# B&R Automation Studio project TD52 (part 60)

#### Gen2_ref.c
```c
/********************************************************************
 * COPYRIGHT -- B&R Industrial Automation GmbH
 ********************************************************************
 * Program: Gen2_ref
 * File: Gen2_ref.c
 * Author: 105055527
 * Last modified by: kelleto00
 * Created: Wed Apr 16 13:02:53 2008
 * Last modified: Wed Oct 09 10:01:33 2024
 * Model Version: 4.14.00.04
 * Description: V4.10.00.01, 01-09-2020 Keller, Ke Estimator, additive LS factor, Ptraj SpeedCtrl, LVRT Freeze HLCi
   V4.10.00.01, 02-10-2020 Keller, bugfix HLCi p2srefLX init, BDC_lib: change Inf to 1e7
   V4.10.00.01, 13-11-2020 Keller, bugfix LXcorr T2s/ZZP, LSLff damping, dbgOut for Leanox WG compensation
   V4.10.00.01, 27-01-2021 Keller, Lx WGV compensation: no reset in island mode, addition before skipfire compensation
   V4.10.00.01, 02-02-2021 Keller, initialization lambda estimation with rLam_Start
   V4.11.00.01, 28-05-2021 Keller, Gas Quality Change (GQC) Improvements, LHV estimator output
   V4.11.00.01, 05-11-2021 Keller, Bugfix BDC: worksplit offset, optionally Nset instead of Nnom, rN_Eng_LRskipF
   V4.12.00.01, 10-02-2021 Keller, SpeedCtrl2.0 TU Wien: Disturbance Estimator, LQR incl. droop & leanox
   V4.12.00.02, 23-05-2022 Arnold, Leanox point C in low load
   V4.12.00.02, 09-06-2022 Kafka, add external skip fire input for isolated and grid parallel operation
   V4.12.00.03, 15-09-2022 Keller, add power trajectory to HLCi for extended LQR (Droop setpoint)
   V4.12.00.04, 12-10-2022 Keller, add gas flow comp. factor for rejections
   V4.12.00.05, 13-10-2022 Keller, power filter for static skipfire in island mode
   V4.12.00.06, 15-11-2022 Keller, Ke adaptation with disturbance observer
   V4.13.00.01, 15-11-2022 Keller, FDC: R_mix output, HLCi: R_mix for Ke
   V4.13.00.02, 10-07-2023 Keller, interpolation of LHV, rho_gas and Lmin
   V4.13.00.03, 10-07-2023 Keller, load dependent gas dosage delay
   V4.13.00.04, 11-09-2023 Keller, D-part FSM, bugfix dPTV ramp
   V4.13.00.05, 27-02-2024 Keller, Filter outputs without bSS
   V4.13.00.06, 10-04-2024 Keller, bugfix leanox manual mode with bSepEmisCtrl
   V4.14.00.01, 01-07-2024 Keller, iNskip_LRfor Ke calculation
   V4.14.00.02, 17-09-2024 Keller, Use actual speed for observer disturbance dg (Gen2_ref/HLC_Island (HLC_Island_ref)/iLQR_SF/Ref LQR)
   V4.14.00.03, 30-09-2024 Keller, LR gas flow compensation possible without actuator saturation
   V4.14.00.04, 02-10-2024 Keller, Limit derivative power setpoint for FSM
 * modified Comment:
 ********************************************************************
 * Implementation of program Gen2_ref
 ********************************************************************
 * Generated with B&R Automation Studio Target for Simulink V6.7.1
 * (ERT based)
 ********************************************************************/

#include "Gen2_ref.h"
#include "Gen2_ref_private.h"

/*  Defines */

/*  Data Types */

/**************************** GLOBAL DATA *************************************/
/*  Definitions */

/*  Declarations  */

/* Forward declaration for local functions */
static real_T Gen2_ref_maximum(const real_T x[13], struct Gen2* inst);

/* Forward declaration for local functions */
static real_T Gen2_ref_minimum(const real_T x[13], struct Gen2* inst);
static real_T Gen2_ref_maximum_f(const real_T x[13], struct Gen2* inst);
static void Gen2_ref_diag(const real_T v[2], real_T d[4], struct Gen2* inst);
static void Gen2_ref_diag_i(const real_T v[4], real_T d[16], struct Gen2* inst);
static void Gen2_ref_diag_i2(const real_T v[3], real_T d[9], struct Gen2* inst);
static void Gen2_ref_state_space_d(const real_T x[3], const real_T p[22], real_T
  Ke_in, real_T Phi[9], real_T h[12], real_T hd[3], struct Gen2* inst);
static void Gen2_ref_diag_i2a(const real_T v[6], real_T d[36], struct Gen2* inst);
static real_T Gen2_ref_det(const real_T x[9], struct Gen2* inst);
static void Gen2_ref_mrdiv(const real_T A[18], const real_T B[9], real_T Y[18], struct Gen2* inst);
static void Gen2_ref_mldivide(const real_T A[16], const real_T B[12], real_T Y
  [12], struct Gen2* inst);
static void Gen2_ref_integrate_model(real_T x0[3], const real_T K[12], const
  real_T u2_past[100], real_T d, const real_T x_disturb[3], const real_T Bd[9],
  real_T x_disturb1_map, const real_T u_sp[4], const real_T x_sp[3], int16_T N,
  const real_T u_min[4], const real_T u_max[4], const real_T p[22], struct Gen2* inst);
static void Gen2_ref_mldivide_j(const real_T A[4], const real_T B[12], real_T Y
  [12], struct Gen2* inst);
static real_T Gen2_ref_maximum_f5(const real_T x[7], struct Gen2* inst);

/***************************** FILE SCOPE DATA ********************************/

/*************************** FUNCTIONS ****************************************/

/* Lookup Binary Search Utility BINARYSEARCH_real_T */
void BINARYSEARCH_real_T(uint32_T *piLeft, uint32_T *piRght, real_T u, const
  real_T *pData, uint32_T iHi, struct Gen2* inst)
{
  /* Find the location of current input value in the data table. */
  *piLeft = 0U;
  *piRght = iHi;
  if (u <= pData[0] ) {
    /* Less than or equal to the smallest point in the table. */
    *piRght = 0U;
  } else if (u >= pData[iHi] ) {
    /* Greater than or equal to the largest point in the table. */
    *piLeft = iHi;
  } else {
    uint32_T i;

    /* Do a binary search. */
    while (( *piRght - *piLeft ) > 1U ) {
      /* Get the average of the left and right indices using to Floor rounding. */
      i = (*piLeft + *piRght) >> 1;

      /* Move either the right index or the left index so that */
      /*  LeftDataPoint <= CurrentValue < RightDataPoint */
      if (u < pData[i] ) {
        *piRght = i;
      } else {
        *piLeft = i;
      }
    }
  }
}

/* Lookup Utility LookUp_real_T_real_T */
void LookUp_real_T_real_T(real_T *pY, const real_T *pYData, real_T u, const
  real_T *pUData, uint32_T iHi, struct Gen2* inst)
{
  uint32_T iLeft;
  uint32_T iRght;
  BINARYSEARCH_real_T( &(iLeft), &(iRght), u, pUData, iHi, inst);

  {
    real_T lambda;
    if (pUData[iRght] > pUData[iLeft] ) {
      real_T num;
      real_T den;
      den = pUData[iRght];
      den -= pUData[iLeft];
      num = u;
      num -= pUData[iLeft];
      lambda = num / den;
    } else {
      lambda = 0.0;
    }

    {
      real_T yLeftCast;
      real_T yRghtCast;
      yLeftCast = pYData[iLeft];
      yRghtCast = pYData[iRght];
      yLeftCast += lambda * ( yRghtCast - yLeftCast );
      (*pY) = yLeftCast;
    }
  }
}

/* Lookup Utility LookUp_real_T_real_T_SAT */
void LookUp_real_T_real_T_SAT(real_T *pY, const real_T *pYData, real_T u, const
  real_T *pUData, uint32_T iHi, struct Gen2* inst)
{
  uint32_T iLeft;
  uint32_T iRght;
  BINARYSEARCH_real_T( &(iLeft), &(iRght), u, pUData, iHi, inst);

  {
    real_T lambda;
    if (pUData[iRght] > pUData[iLeft] ) {
      real_T num;
      real_T den;
      den = pUData[iRght];
      den -= pUData[iLeft];
      num = u;
      num -= pUData[iLeft];
      lambda = num / den;
    } else {
      lambda = 0.0;
    }

    {
      real_T yLeftCast;
      real_T yRghtCast;
      yLeftCast = pYData[iLeft];
      yRghtCast = pYData[iRght];
      yLeftCast += lambda * ( yRghtCast - yLeftCast );
      (*pY) = yLeftCast;
    }
  }
}

/* Lookup Utility LookUp_real_Treal32_T_K4km1JJi */
void LookUp_real_Treal32_T_K4km1JJi(real_T *pY, const real32_T *pYData, real_T
  u, const real_T *pUData, uint32_T iHi, struct Gen2* inst)
{
  uint32_T iLeft;
  uint32_T iRght;
  BINARYSEARCH_real_T( &(iLeft), &(iRght), u, pUData, iHi, inst);

  {
    real_T lambda;
    if (pUData[iRght] > pUData[iLeft] ) {
      real_T num;
      real_T den;
      den = pUData[iRght];
      den -= pUData[iLeft];
      num = u;
      num -= pUData[iLeft];
      lambda = num / den;
    } else {
      lambda = 0.0;
    }

    {
      real_T yLeftCast;
      real_T yRghtCast;
      yLeftCast = pYData[iLeft];
      yRghtCast = pYData[iRght];
      yLeftCast += lambda * ( yRghtCast - yLeftCast );
      (*pY) = yLeftCast;
    }
  }
}

/* Lookup Binary Search Utility BINARYSEARCH_real32_Treal_T */
void BINARYSEARCH_real32_Treal_T(uint32_T *piLeft, uint32_T *piRght, real32_T u,
  const real_T *pData, uint32_T iHi, struct Gen2* inst)
{
  real_T uCast;

  /* cast current input to the data type/scaling of the table data */
  uCast = u;

  /* Find the location of current input value in the data table. */
  *piLeft = 0U;
  *piRght = iHi;
  if (uCast < pData[0] ) {
    /* Less than the smallest point in the table. */
    *piRght = 0U;
  } else if (uCast >= pData[iHi] ) {
    /* Greater than or equal to the largest point in the table. */
    *piLeft = iHi;
  } else {
    uint32_T i;

    /* Do a binary search. */
    while (( *piRght - *piLeft ) > 1U ) {
      /* Get the average of the left and right indices using to Floor rounding. */
      i = (*piLeft + *piRght) >> 1;

      /* Move either the right index or the left index so that */
      /*  LeftDataPoint <= CurrentValue < RightDataPoint */
      if (uCast < pData[i] ) {
        *piRght = i;
      } else {
        *piLeft = i;
      }
    }
  }
}

/* Lookup Utility LookUp_real_T_real32_Treal_T */
void LookUp_real_T_real32_Treal_T(real_T *pY, const real_T *pYData, real32_T u,
  const real_T *pUData, uint32_T iHi, struct Gen2* inst)
{
  uint32_T iLeft;
  uint32_T iRght;
  BINARYSEARCH_real32_Treal_T( &(iLeft), &(iRght), u, pUData, iHi, inst);

  {
    real_T lambda;
    if (pUData[iRght] > pUData[iLeft] ) {
      real_T num;
      real_T den;
      den = pUData[iRght];
      den -= pUData[iLeft];
      num = u;
      num -= pUData[iLeft];
      lambda = num / den;
    } else {
      lambda = 0.0;
    }

    {
      real_T yLeftCast;
      real_T yRghtCast;
      yLeftCast = pYData[iLeft];
      yRghtCast = pYData[iRght];
      yLeftCast += lambda * ( yRghtCast - yLeftCast );
      (*pY) = yLeftCast;
    }
  }
}

real_T look1_binlxpw(real_T u0, const real_T bp0[], const real_T table[],
                     uint32_T maxIndex, struct Gen2* inst)
{
  real_T frac;
  real_T yL_0d0;
  uint32_T bpIdx;
  uint32_T iLeft;
  uint32_T iRght;

  /* Column-major Lookup 1-D
     Search method: 'binary'
     Use previous index: 'off'
     Interpolation method: 'Linear point-slope'
     Extrapolation method: 'Linear'
     Use last breakpoint for index at or above upper limit: 'off'
     Remove protection against out-of-range input in generated code: 'off'
   */
  /* Prelookup - Index and Fraction
     Index Search method: 'binary'
     Extrapolation method: 'Linear'
     Use previous index: 'off'
     Use last breakpoint for index at or above upper limit: 'off'
     Remove protection against out-of-range input in generated code: 'off'
   */
  if (u0 <= bp0[0U]) {
    iLeft = 0U;
    frac = (u0 - bp0[0U]) / (bp0[1U] - bp0[0U]);
  } else if (u0 < bp0[maxIndex]) {
    /* Binary Search */
    bpIdx = maxIndex >> 1U;
    iLeft = 0U;
    iRght = maxIndex;
    while (iRght - iLeft > 1U) {
      if (u0 < bp0[bpIdx]) {
        iRght = bpIdx;
      } else {
        iLeft = bpIdx;
      }

      bpIdx = (iRght + iLeft) >> 1U;
    }

    frac = (u0 - bp0[iLeft]) / (bp0[iLeft + 1U] - bp0[iLeft]);
  } else {
    iLeft = maxIndex - 1U;
    frac = (u0 - bp0[maxIndex - 1U]) / (bp0[maxIndex] - bp0[maxIndex - 1U]);
  }

  /* Column-major Interpolation 1-D
     Interpolation method: 'Linear point-slope'
     Use last breakpoint for index at or above upper limit: 'off'
     Overflow mode: 'portable wrapping'
   */
  yL_0d0 = table[iLeft];
  return (table[iLeft + 1U] - yL_0d0) * frac + yL_0d0;
}

/*
 * System initialize for atomic system:
 *    '<S23>/Filter1'
 *    '<S23>/Filter2'
 *    '<S23>/Filter4'
 *    '<S344>/WO1'
 *    '<S424>/Filter1'
 */
void Gen2_ref_Filter1_Init(rtDW_Filter1_Gen2_ref *localDW, struct Gen2* inst)
{
  /* InitializeConditions for DiscreteIntegrator: '<S49>/Discrete-Time Integrator' */
  localDW->DiscreteTimeIntegrator_IC_LOADI = 1U;
}

/*
 * Output and update for atomic system:
 *    '<S23>/Filter1'
 *    '<S23>/Filter2'
 *    '<S23>/Filter4'
 *    '<S344>/WO1'
 *    '<S424>/Filter1'
 */
void Gen2_ref_Filter1(real_T rtu_in, real_T rtu_T_filt, boolean_T rtu_reset,
                      rtB_Filter1_Gen2_ref *localB, rtDW_Filter1_Gen2_ref
                      *localDW, struct Gen2* inst)
{
  real_T rtb_Divide4_p;
  boolean_T rtb_LogicalOperator_kj;

  /* Logic: '<S49>/Logical Operator' incorporates:
   *  Constant: '<S49>/Constant'
   *  Logic: '<S49>/Logical Operator1'
   *  RelationalOperator: '<S49>/Relational Operator'
   */
  rtb_LogicalOperator_kj = (rtu_reset || (!(rtu_T_filt > 0.0)));

  /* DiscreteIntegrator: '<S49>/Discrete-Time Integrator' */
  if (localDW->DiscreteTimeIntegrator_IC_LOADI != 0) {
    localDW->DiscreteTimeIntegrator_DSTATE = rtu_in;
  }

  if (rtb_LogicalOperator_kj || (localDW->DiscreteTimeIntegrator_PrevRese != 0))
  {
    localDW->DiscreteTimeIntegrator_DSTATE = rtu_in;
  }

  /* Switch: '<S71>/Switch' incorporates:
   *  Abs: '<S71>/Abs'
   *  Constant: '<S71>/Constant2'
   *  RelationalOperator: '<S71>/Relational Operator'
   */
  if (2.2204460492503131E-16 >= fabs(rtu_T_filt)) {
    rtb_Divide4_p = 2.2204460492503131E-16;
  } else {
    rtb_Divide4_p = rtu_T_filt;
  }

  /* End of Switch: '<S71>/Switch' */

  /* Product: '<S49>/Divide4' incorporates:
   *  DiscreteIntegrator: '<S49>/Discrete-Time Integrator'
   *  Sum: '<S49>/Sum4'
   */
  rtb_Divide4_p = (rtu_in - localDW->DiscreteTimeIntegrator_DSTATE) /
    rtb_Divide4_p;

  /* Switch: '<S49>/Switch1' */
  if (rtb_LogicalOperator_kj) {
    /* Switch: '<S49>/Switch1' incorporates:
     *  Constant: '<S49>/Constant'
     */
    localB->Switch1 = 0.0;
  } else {
    /* Switch: '<S49>/Switch1' */
    localB->Switch1 = rtb_Divide4_p;
  }

  /* End of Switch: '<S49>/Switch1' */

  /* Update for DiscreteIntegrator: '<S49>/Discrete-Time Integrator' */
  localDW->DiscreteTimeIntegrator_IC_LOADI = 0U;
  localDW->DiscreteTimeIntegrator_DSTATE += 0.01 * rtb_Divide4_p;
  localDW->DiscreteTimeIntegrator_PrevRese = (int8_T)rtb_LogicalOperator_kj;
}

/*
 * Output and update for atomic system:
 *    '<S23>/TON_1'
 *    '<S6>/TON'
 *    '<S667>/TON1'
 *    '<S634>/Delay Retard'
 *    '<S634>/TON'
 *    '<S714>/TON'
 *    '<S715>/TON'
 *    '<S716>/TON'
 *    '<S747>/TON'
 *    '<S831>/TON1'
 *    ...
 */
void Gen2_ref_TON_1(boolean_T rtu_IN, real_T rtu_PT, rtB_TON_1_Gen2_ref *localB,
                    rtDW_TON_1_Gen2_ref *localDW, struct Gen2* inst)
{
  boolean_T rtb_LogicalOperator2_oe;
  boolean_T rtb_RelationalOperator_m1;

  /* Logic: '<S61>/Logical Operator2' */
  rtb_LogicalOperator2_oe = !rtu_IN;

  /* DiscreteIntegrator: '<S61>/Discrete-Time Integrator' */
  if (rtb_LogicalOperator2_oe || (localDW->DiscreteTimeIntegrator_PrevRese != 0))
  {
    localDW->DiscreteTimeIntegrator_DSTATE = 0.0;
  }

  /* RelationalOperator: '<S61>/Relational Operator' incorporates:
   *  DiscreteIntegrator: '<S61>/Discrete-Time Integrator'
   */
  rtb_RelationalOperator_m1 = (localDW->DiscreteTimeIntegrator_DSTATE >= rtu_PT);

  /* Logic: '<S61>/Logical Operator3' */
  localB->LogicalOperator3 = (rtb_RelationalOperator_m1 && rtu_IN);

  /* Update for DiscreteIntegrator: '<S61>/Discrete-Time Integrator' incorporates:
   *  DataTypeConversion: '<S95>/Conversion'
   *  Logic: '<S61>/Logical Operator'
   *  Logic: '<S61>/Logical Operator1'
   */
  localDW->DiscreteTimeIntegrator_DSTATE += (real_T)((!rtb_RelationalOperator_m1)
    && rtu_IN) * 0.01;
  localDW->DiscreteTimeIntegrator_PrevRese = (int8_T)rtb_LogicalOperator2_oe;
}

/*
 * System initialize for atomic system:
 *    '<S62>/Filter3'
 *    '<S134>/Filter'
 *    '<S344>/WO2'
 *    '<S585>/Filter'
 *    '<S628>/Filter'
 *    '<S633>/Filter'
 *    '<S761>/Filter1'
 *    '<S19>/Filter'
 *    '<S19>/Filter1'
 *    '<S20>/Filter'
 *    ...
 */
void Gen2_ref_Filter3_Init(real_T rtu_x0, rtDW_Filter3_Gen2_ref *localDW, struct Gen2* inst)
{
  /* InitializeConditions for DiscreteIntegrator: '<S97>/Discrete-Time Integrator' */
  localDW->DiscreteTimeIntegrator_DSTATE = rtu_x0;
}

/*
 * Output and update for atomic system:
 *    '<S62>/Filter3'
 *    '<S134>/Filter'
 *    '<S344>/WO2'
 *    '<S585>/Filter'
 *    '<S628>/Filter'
 *    '<S633>/Filter'
 *    '<S761>/Filter1'
 *    '<S19>/Filter'
 *    '<S19>/Filter1'
 *    '<S20>/Filter'
 *    ...
 */
void Gen2_ref_Filter3(real_T rtu_in, real_T rtu_T_filt, real_T rtu_x0, boolean_T
                      rtu_reset, rtB_Filter3_Gen2_ref *localB,
                      rtDW_Filter3_Gen2_ref *localDW, struct Gen2* inst)
{
  real_T tmp;
  boolean_T rtb_LogicalOperator_hy;
  boolean_T rtb_RelationalOperator_hc;

  /* RelationalOperator: '<S97>/Relational Operator' incorporates:
   *  Constant: '<S97>/Constant'
   */
  rtb_RelationalOperator_hc = (rtu_T_filt > 0.0);

  /* Logic: '<S97>/Logical Operator' incorporates:
   *  Logic: '<S97>/Logical Operator1'
   */
  rtb_LogicalOperator_hy = (rtu_reset || (!rtb_RelationalOperator_hc));

  /* DiscreteIntegrator: '<S97>/Discrete-Time Integrator' */
  if (rtb_LogicalOperator_hy || (localDW->DiscreteTimeIntegrator_PrevRese != 0))
  {
    localDW->DiscreteTimeIntegrator_DSTATE = rtu_x0;
  }

  /* Switch: '<S97>/Switch' */
  if (rtb_RelationalOperator_hc) {
    /* Switch: '<S97>/Switch' incorporates:
     *  DiscreteIntegrator: '<S97>/Discrete-Time Integrator'
     */
    localB->Switch = localDW->DiscreteTimeIntegrator_DSTATE;
  } else {
    /* Switch: '<S97>/Switch' */
    localB->Switch = rtu_in;
  }

  /* End of Switch: '<S97>/Switch' */

  /* Switch: '<S100>/Switch' incorporates:
   *  Abs: '<S100>/Abs'
   *  Constant: '<S100>/Constant2'
   *  RelationalOperator: '<S100>/Relational Operator'
   */
  if (2.2204460492503131E-16 >= fabs(rtu_T_filt)) {
    tmp = 2.2204460492503131E-16;
  } else {
    tmp = rtu_T_filt;
  }

  /* End of Switch: '<S100>/Switch' */

  /* Update for DiscreteIntegrator: '<S97>/Discrete-Time Integrator' incorporates:
   *  Product: '<S97>/Divide4'
   *  Sum: '<S97>/Sum4'
   */
  localDW->DiscreteTimeIntegrator_DSTATE += (rtu_in -
    localDW->DiscreteTimeIntegrator_DSTATE) / tmp * 0.01;
  localDW->DiscreteTimeIntegrator_PrevRese = (int8_T)rtb_LogicalOperator_hy;
}

/*
 * System initialize for atomic system:
 *    '<S24>/MATLAB Function'
 *    '<S25>/MATLAB Function'
 */
void Gen2_ref_MATLABFunction_Init(rtDW_MATLABFunction_Gen2_ref *localDW, struct Gen2* inst)
{
  localDW->out = 2.0;
}

/*
 * Output and update for atomic system:
 *    '<S24>/MATLAB Function'
 *    '<S25>/MATLAB Function'
 */
void Gen2_ref_MATLABFunction(real_T rtu_u, real_T rtu_u_deact, real_T rtu_u_act,
  rtB_MATLABFunction_Gen2_ref *localB, rtDW_MATLABFunction_Gen2_ref *localDW, struct Gen2* inst)
{
  if (rtu_u > rtu_u_act) {
    localDW->out = 1.0;
  } else if (rtu_u < rtu_u_deact) {
    localDW->out = 2.0;
  }

  localB->y = localDW->out;
}

/*
 * Output and update for atomic system:
 *    '<S27>/engine massflow'
 *    '<S46>/engine massflow'
 */
void Gen2_ref_enginemassflow(real_T rtu_p_2s, real_T rtu_T_2s, real_T rtu_n_e,
  real_T rtu_eta_V, real_T rtu_V_d, rtB_enginemassflow_Gen2_ref *localB, struct Gen2* inst)
{
  real_T u0;
  u0 = 287.15 * rtu_T_2s;
  if (!(u0 >= 1.0)) {
    u0 = 1.0;
  }

  localB->dm_e = rtu_eta_V * rtu_V_d * rtu_p_2s / u0 * rtu_n_e / 2.0 /
    6.2831853071795862;
}

/*
 * Output and update for atomic system:
 *    '<S1>/IntegerZOH'
 *    '<S1>/IntegerZOH2'
 *    '<S5>/IntegerZOH'
 *    '<S5>/IntegerZOH1'
 *    '<S8>/IntegerZOH'
 */
void Gen2_ref_IntegerZOH(real_T rtu_u, int16_T rtu_i, rtB_IntegerZOH_Gen2_ref
  *localB, rtDW_IntegerZOH_Gen2_ref *localDW, struct Gen2* inst)
{
  if (!localDW->count_not_empty) {
    localDW->count_not_empty = true;
    localDW->u_z = rtu_u;
  }

  if (localDW->count < rtu_i) {
    localB->y = localDW->u_z;
    localDW->count++;
  } else {
    localB->y = rtu_u;
    localDW->u_z = rtu_u;
    localDW->count = 1.0;
  }
}

/*
 * Output and update for atomic system:
 *    '<S144>/lam2cg1'
 *    '<S267>/lam2cg'
 *    '<S268>/lam2cg'
 */
void Gen2_ref_lam2cg1(real_T rtu_lam, real_T rtu_AFRs, rtB_lam2cg1_Gen2_ref
                      *localB, struct Gen2* inst)
{
  real_T rtb_Switch_oai;

  /* Bias: '<S150>/Bias' incorporates:
   *  Product: '<S150>/Product'
   */
  rtb_Switch_oai = rtu_lam * rtu_AFRs + 1.0;

  /* Switch: '<S152>/Switch' incorporates:
   *  Abs: '<S152>/Abs'
   *  Constant: '<S152>/Constant2'
   *  RelationalOperator: '<S152>/Relational Operator'
   */
  if (2.2204460492503131E-16 >= fabs(rtb_Switch_oai)) {
    rtb_Switch_oai = 2.2204460492503131E-16;
  }

  /* End of Switch: '<S152>/Switch' */

  /* Product: '<S150>/Divide' incorporates:
   *  Constant: '<S150>/Constant'
   */
  localB->Divide = 1.0 / rtb_Switch_oai;
}

/*
 * Output and update for atomic system:
 *    '<S44>/engine massflow2'
 *    '<S46>/engine massflow1'
 */
void Gen2_ref_enginemassflow2(real_T rtu_p_2s, real_T rtu_T_2s, real_T rtu_n_e,
  real_T rtu_eta_V, real_T rtu_V_d, rtB_enginemassflow2_Gen2_ref *localB, struct Gen2* inst)
{
  real_T u0;
  u0 = 287.15 * rtu_T_2s;
  if (!(u0 >= 1.0)) {
    u0 = 1.0;
  }

  localB->dm_e = rtu_eta_V * rtu_V_d * rtu_p_2s / u0 * rtu_n_e / 2.0 /
    6.2831853071795862;
}

/*
 * Output and update for atomic system:
 *    '<S161>/Inverse_Linearization4'
 *    '<S45>/Inverse_Linearization1'
 *    '<S45>/Inverse_Linearization3'
 *    '<S45>/Inverse_Linearization2'
 */
void Gen2_ref_Inverse_Linearization4(real_T rtu_rPos_TV_u, const tGen2Parameter *
  rtu_rPos_TV_u_f, rtB_Inverse_Linearization4_Gen2 *localB, struct Gen2* inst)
{
  /* S-Function (sfix_look1_dyn): '<S169>/LCRScal_Lam_EOT1' */
  /* Dynamic Look-Up Table Block: '<S169>/LCRScal_Lam_EOT1'
   * Input0  Data Type:  Floating Point real_T
   * Input1  Data Type:  Floating Point real_T
   * Input2  Data Type:  Floating Point real_T
   * Output0 Data Type:  Floating Point real_T
   * Lookup Method: Linear_Endpoint
   *
   */
  LookUp_real_T_real_T( &(localB->LCRScal_Lam_EOT1),
                       &rtu_rPos_TV_u_f->bdcTv.rPosTv_Lin_x[0], rtu_rPos_TV_u,
                       &rtu_rPos_TV_u_f->bdcTv.rPosTv_Lin_y[0], 9U, inst);
}

/*
 * System initialize for atomic system:
 *    '<S190>/N_TC_HP_filt'
 *    '<S192>/N_TC_LP_filt'
 *    '<S193>/N_TC_LP_filt'
 *    '<S194>/Pel_filt'
 *    '<S195>/T1HP_filt'
 *    '<S196>/T1LP_filt'
 *    '<S197>/T2s_filt'
 *    '<S201>/Volt_filt'
 *    '<S202>/p1HP_filt'
 *    '<S204>/p2HP_filt'
 *    ...
 */
void Gen2_ref_N_TC_HP_filt_Init(rtDW_N_TC_HP_filt_Gen2_ref *localDW, struct Gen2* inst)
{
  /* InitializeConditions for DiscreteIntegrator: '<S209>/Discrete-Time Integrator' */
  localDW->DiscreteTimeIntegrator_IC_LOADI = 1U;
}

/*
 * Output and update for atomic system:
 *    '<S190>/N_TC_HP_filt'
 *    '<S192>/N_TC_LP_filt'
 *    '<S193>/N_TC_LP_filt'
 *    '<S194>/Pel_filt'
 *    '<S195>/T1HP_filt'
 *    '<S196>/T1LP_filt'
 *    '<S197>/T2s_filt'
 *    '<S201>/Volt_filt'
 *    '<S202>/p1HP_filt'
 *    '<S204>/p2HP_filt'
 *    ...
 */
void Gen2_ref_N_TC_HP_filt(real_T rtu_in, real_T rtu_T_filt, boolean_T rtu_reset,
  rtB_N_TC_HP_filt_Gen2_ref *localB, rtDW_N_TC_HP_filt_Gen2_ref *localDW, struct Gen2* inst)
{
  real_T tmp;
  boolean_T rtb_LogicalOperator_ip;
  boolean_T rtb_RelationalOperator_glm;

  /* RelationalOperator: '<S209>/Relational Operator' incorporates:
   *  Constant: '<S209>/Constant'
   */
  rtb_RelationalOperator_glm = (rtu_T_filt > 0.0);

  /* Logic: '<S209>/Logical Operator' incorporates:
   *  Logic: '<S209>/Logical Operator1'
   */
  rtb_LogicalOperator_ip = (rtu_reset || (!rtb_RelationalOperator_glm));

  /* DiscreteIntegrator: '<S209>/Discrete-Time Integrator' */
  if (localDW->DiscreteTimeIntegrator_IC_LOADI != 0) {
    localDW->DiscreteTimeIntegrator_DSTATE = rtu_in;
  }

  if (rtb_LogicalOperator_ip || (localDW->DiscreteTimeIntegrator_PrevRese != 0))
  {
    localDW->DiscreteTimeIntegrator_DSTATE = rtu_in;
  }

  /* Switch: '<S209>/Switch' */
  if (rtb_RelationalOperator_glm) {
    /* Switch: '<S209>/Switch' incorporates:
     *  DiscreteIntegrator: '<S209>/Discrete-Time Integrator'
     */
    localB->Switch = localDW->DiscreteTimeIntegrator_DSTATE;
  } else {
    /* Switch: '<S209>/Switch' */
    localB->Switch = rtu_in;
  }

  /* End of Switch: '<S209>/Switch' */

  /* Update for DiscreteIntegrator: '<S209>/Discrete-Time Integrator' */
  localDW->DiscreteTimeIntegrator_IC_LOADI = 0U;

  /* Switch: '<S210>/Switch' incorporates:
   *  Abs: '<S210>/Abs'
   *  Constant: '<S210>/Constant2'
   *  RelationalOperator: '<S210>/Relational Operator'
   */
  if (2.2204460492503131E-16 >= fabs(rtu_T_filt)) {
    tmp = 2.2204460492503131E-16;
  } else {
    tmp = rtu_T_filt;
  }

  /* End of Switch: '<S210>/Switch' */

  /* Update for DiscreteIntegrator: '<S209>/Discrete-Time Integrator' incorporates:
   *  Product: '<S209>/Divide4'
   *  Sum: '<S209>/Sum4'
   */
  localDW->DiscreteTimeIntegrator_DSTATE += (rtu_in -
    localDW->DiscreteTimeIntegrator_DSTATE) / tmp * 0.01;
  localDW->DiscreteTimeIntegrator_PrevRese = (int8_T)rtb_LogicalOperator_ip;
}

/*
 * Output and update for atomic system:
 *    '<S267>/Mg'
 *    '<S268>/Mg'
 */
void Gen2_ref_Mg(real_T rtu_rhoGas, rtB_Mg_Gen2_ref *localB, struct Gen2* inst)
{
  real_T tmp;

  /* Switch: '<S279>/Switch' incorporates:
   *  Abs: '<S279>/Abs'
   *  Constant: '<S279>/Constant2'
   *  RelationalOperator: '<S279>/Relational Operator'
   */
  if (2.2204460492503131E-16 >= fabs(rtu_rhoGas)) {
    tmp = 2.2204460492503131E-16;
  } else {
    tmp = rtu_rhoGas;
  }

  /* End of Switch: '<S279>/Switch' */

  /* Bias: '<S274>/Bias' incorporates:
   *  Constant: '<S274>/rhoAir'
   *  Product: '<S274>/Divide'
   */
  localB->Bias = 1.293 / tmp + -1.0;
}

/*
 * Output and update for atomic system:
 *    '<S267>/lam2cg1'
 *    '<S268>/lam2cg1'
 */
void Gen2_ref_lam2cg1_a(real_T rtu_lam, real_T rtu_Lmin, rtB_lam2cg1_Gen2_ref_i *
  localB, struct Gen2* inst)
{
  real_T rtb_Switch_nb;

  /* Bias: '<S277>/Bias' incorporates:
   *  Product: '<S277>/Product'
   */
  rtb_Switch_nb = rtu_lam * rtu_Lmin + 1.0;

  /* Switch: '<S287>/Switch' incorporates:
   *  Abs: '<S287>/Abs'
   *  Constant: '<S287>/Constant2'
   *  RelationalOperator: '<S287>/Relational Operator'
   */
  if (2.2204460492503131E-16 >= fabs(rtb_Switch_nb)) {
    rtb_Switch_nb = 2.2204460492503131E-16;
  }

  /* End of Switch: '<S287>/Switch' */

  /* Product: '<S277>/Divide' incorporates:
   *  Constant: '<S277>/Constant'
   */
  localB->Divide = 1.0 / rtb_Switch_nb;
}

/*
 * Output and update for atomic system:
 *    '<S305>/FILTER no delay'
 *    '<S305>/FILTER no delay1'
 *    '<S305>/FILTER no delay2'
 *    '<S305>/FILTER no delay3'
 *    '<S305>/FILTER no delay4'
 *    '<S305>/FILTER no delay5'
 *    '<S628>/FILTER no delay'
 */
void Gen2_ref_FILTERnodelay(real_T rtu_u, real_T rtu_T, real_T rtu_Ts, boolean_T
  rtu_reset, rtB_FILTERnodelay_Gen2_ref *localB, rtDW_FILTERnodelay_Gen2_ref
  *localDW, struct Gen2* inst)
{
  real_T d_dt;
  if ((!localDW->x_not_empty) || rtu_reset) {
    localDW->x = rtu_u;
    localDW->x_not_empty = true;
  }

  if (rtu_Ts > 0.0) {
    if (rtu_T >= rtu_Ts) {
      d_dt = rtu_T;
    } else {
      d_dt = rtu_Ts;
    }

    d_dt = (rtu_u - localDW->x) / d_dt;
    localDW->x += rtu_Ts * d_dt;
    localB->y = localDW->x;
  } else {
    d_dt = rtu_u - localDW->x;
    localDW->x = rtu_u;
    localB->y = rtu_u;
  }

  localB->d_dt = d_dt;
}

/*
 * System initialize for atomic system:
 *    '<S306>/2nd Order Filter'
 *    '<S306>/2nd Order Filter1'
 *    '<S306>/2nd Order Filter2'
 */
void Gen2_ref_undOrderFilter_Init(rtDW_undOrderFilter_Gen2_ref *localDW, struct Gen2* inst)
{
  /* InitializeConditions for DiscreteIntegrator: '<S314>/Discrete-Time Integrator1' */
  localDW->DiscreteTimeIntegrator1_IC_LOAD = 1U;
}

/*
 * Output and update for atomic system:
 *    '<S306>/2nd Order Filter'
 *    '<S306>/2nd Order Filter1'
 *    '<S306>/2nd Order Filter2'
 */
void Gen2_ref_undOrderFilter(real_T rtu_in, real_T rtu_omega, real_T rtu_d,
  boolean_T rtu_reset, rtB_undOrderFilter_Gen2_ref *localB,
  rtDW_undOrderFilter_Gen2_ref *localDW, struct Gen2* inst)
{
  real_T rtb_Divide1_jr;
  real_T rtb_a0b0_o;
  real_T rtb_x2_g;

  /* DiscreteIntegrator: '<S314>/Discrete-Time Integrator' */
  if (rtu_reset || (localDW->DiscreteTimeIntegrator_PrevRese != 0)) {
    localDW->DiscreteTimeIntegrator_DSTATE = 0.0;
  }

  rtb_x2_g = localDW->DiscreteTimeIntegrator_DSTATE;

  /* Product: '<S314>/Product' */
  rtb_a0b0_o = rtu_omega * rtu_omega;

  /* Switch: '<S319>/Switch' incorporates:
   *  Abs: '<S319>/Abs'
   *  Constant: '<S319>/Constant2'
   *  RelationalOperator: '<S319>/Relational Operator'
   */
  if (2.2204460492503131E-16 >= fabs(rtb_a0b0_o)) {
    rtb_Divide1_jr = 2.2204460492503131E-16;
  } else {
    rtb_Divide1_jr = rtb_a0b0_o;
  }

  /* End of Switch: '<S319>/Switch' */

  /* Product: '<S314>/Divide1' */
  rtb_Divide1_jr = rtu_in / rtb_Divide1_jr;

  /* DiscreteIntegrator: '<S314>/Discrete-Time Integrator1' */
  if (localDW->DiscreteTimeIntegrator1_IC_LOAD != 0) {
    localDW->DiscreteTimeIntegrator1_DSTATE = rtb_Divide1_jr;
  }

  if (rtu_reset || (localDW->DiscreteTimeIntegrator1_PrevRes != 0)) {
    localDW->DiscreteTimeIntegrator1_DSTATE = rtb_Divide1_jr;
  }

  /* Switch: '<S314>/Switch1' incorporates:
   *  RelationalOperator: '<S314>/Relational Operator'
   */
  if (rtb_a0b0_o > 0.0) {
    /* Switch: '<S314>/Switch1' incorporates:
     *  DiscreteIntegrator: '<S314>/Discrete-Time Integrator'
     *  Product: '<S314>/Product5'
     */
    localB->Switch1 = rtb_a0b0_o * localDW->DiscreteTimeIntegrator_DSTATE;
  } else {
    /* Switch: '<S314>/Switch1' */
    localB->Switch1 = 0.0;
  }

  /* End of Switch: '<S314>/Switch1' */

  /* Update for DiscreteIntegrator: '<S314>/Discrete-Time Integrator' incorporates:
   *  Constant: '<S314>/Constant1'
   *  DiscreteIntegrator: '<S314>/Discrete-Time Integrator1'
   *  Product: '<S314>/Product1'
   *  Product: '<S314>/Product3'
   *  Product: '<S314>/Product4'
   *  Sum: '<S314>/Sum'
   */
  localDW->DiscreteTimeIntegrator_DSTATE += ((rtu_in - rtb_a0b0_o *
    localDW->DiscreteTimeIntegrator1_DSTATE) - rtu_omega * rtu_d * 2.0 *
    localDW->DiscreteTimeIntegrator_DSTATE) * 0.01;
  localDW->DiscreteTimeIntegrator_PrevRese = (int8_T)rtu_reset;

  /* Update for DiscreteIntegrator: '<S314>/Discrete-Time Integrator1' incorporates:
   *  DiscreteIntegrator: '<S314>/Discrete-Time Integrator'
   */
  localDW->DiscreteTimeIntegrator1_IC_LOAD = 0U;
  localDW->DiscreteTimeIntegrator1_DSTATE += 0.01 * rtb_x2_g;
  localDW->DiscreteTimeIntegrator1_PrevRes = (int8_T)rtu_reset;
}

/*
 * System initialize for atomic system:
 *    '<S306>/2nd Order Filter3'
 *    '<S418>/2nd Order Filter'
 */
void Gen2_ref_undOrderFilter3_Init(rtDW_undOrderFilter3_Gen2_ref *localDW, struct Gen2* inst)
{
  /* InitializeConditions for DiscreteIntegrator: '<S317>/Discrete-Time Integrator1' */
  localDW->DiscreteTimeIntegrator1_IC_LOAD = 1U;
}

/*
 * Output and update for atomic system:
 *    '<S306>/2nd Order Filter3'
 *    '<S418>/2nd Order Filter'
 */
void Gen2_ref_undOrderFilter3(real_T rtu_in, real_T rtu_omega, real_T rtu_d,
  boolean_T rtu_reset, rtB_undOrderFilter3_Gen2_ref *localB,
  rtDW_undOrderFilter3_Gen2_ref *localDW, struct Gen2* inst)
{
  real_T rtb_Divide1_k;
  real_T rtb_a0b0_e;
  real_T rtb_x2_f;

  /* DiscreteIntegrator: '<S317>/Discrete-Time Integrator' */
  if (rtu_reset || (localDW->DiscreteTimeIntegrator_PrevRese != 0)) {
    localDW->DiscreteTimeIntegrator_DSTATE = 0.0;
  }

  rtb_x2_f = localDW->DiscreteTimeIntegrator_DSTATE;

  /* Product: '<S317>/Product' */
  rtb_a0b0_e = rtu_omega * rtu_omega;

  /* Switch: '<S325>/Switch' incorporates:
   *  Abs: '<S325>/Abs'
   *  Constant: '<S325>/Constant2'
   *  RelationalOperator: '<S325>/Relational Operator'
   */
  if (2.2204460492503131E-16 >= fabs(rtb_a0b0_e)) {
    rtb_Divide1_k = 2.2204460492503131E-16;
  } else {
    rtb_Divide1_k = rtb_a0b0_e;
  }

  /* End of Switch: '<S325>/Switch' */

  /* Product: '<S317>/Divide1' */
  rtb_Divide1_k = rtu_in / rtb_Divide1_k;

  /* DiscreteIntegrator: '<S317>/Discrete-Time Integrator1' */
  if (localDW->DiscreteTimeIntegrator1_IC_LOAD != 0) {
    localDW->DiscreteTimeIntegrator1_DSTATE = rtb_Divide1_k;
  }

  if (rtu_reset || (localDW->DiscreteTimeIntegrator1_PrevRes != 0)) {
    localDW->DiscreteTimeIntegrator1_DSTATE = rtb_Divide1_k;
  }

  /* Switch: '<S317>/Switch' incorporates:
   *  RelationalOperator: '<S317>/Relational Operator'
   *  Switch: '<S317>/Switch1'
   */
  if (rtb_a0b0_e > 0.0) {
    /* Switch: '<S317>/Switch' incorporates:
     *  DiscreteIntegrator: '<S317>/Discrete-Time Integrator1'
     *  Product: '<S317>/Product2'
     */
    localB->Switch = localDW->DiscreteTimeIntegrator1_DSTATE * rtb_a0b0_e;

    /* Switch: '<S317>/Switch1' incorporates:
     *  DiscreteIntegrator: '<S317>/Discrete-Time Integrator'
     *  Product: '<S317>/Product5'
     */
    localB->Switch1 = rtb_a0b0_e * localDW->DiscreteTimeIntegrator_DSTATE;
  } else {
    /* Switch: '<S317>/Switch' */
    localB->Switch = rtu_in;

    /* Switch: '<S317>/Switch1' */
    localB->Switch1 = 0.0;
  }

  /* End of Switch: '<S317>/Switch' */

  /* Update for DiscreteIntegrator: '<S317>/Discrete-Time Integrator' incorporates:
   *  Constant: '<S317>/Constant1'
   *  DiscreteIntegrator: '<S317>/Discrete-Time Integrator1'
   *  Product: '<S317>/Product1'
   *  Product: '<S317>/Product3'
   *  Product: '<S317>/Product4'
   *  Sum: '<S317>/Sum'
   */
  localDW->DiscreteTimeIntegrator_DSTATE += ((rtu_in - rtb_a0b0_e *
    localDW->DiscreteTimeIntegrator1_DSTATE) - rtu_omega * rtu_d * 2.0 *
    localDW->DiscreteTimeIntegrator_DSTATE) * 0.01;
  localDW->DiscreteTimeIntegrator_PrevRese = (int8_T)rtu_reset;

  /* Update for DiscreteIntegrator: '<S317>/Discrete-Time Integrator1' incorporates:
   *  DiscreteIntegrator: '<S317>/Discrete-Time Integrator'
   */
  localDW->DiscreteTimeIntegrator1_IC_LOAD = 0U;
  localDW->DiscreteTimeIntegrator1_DSTATE += 0.01 * rtb_x2_f;
  localDW->DiscreteTimeIntegrator1_PrevRes = (int8_T)rtu_reset;
}

/*
 * System initialize for atomic system:
 *    '<S6>/TOF'
 *    '<S6>/TOF1'
 *    '<S6>/TOF2'
 *    '<S425>/TOF'
 *    '<S427>/TOF1'
 *    '<S427>/TOF3'
 *    '<S667>/TOF'
 *    '<S831>/TOF'
 */
void Gen2_ref_TOF_Init(rtDW_TOF_Gen2_ref *localDW, struct Gen2* inst)
{
  /* InitializeConditions for DiscreteIntegrator: '<S329>/Discrete-Time Integrator' */
  localDW->DiscreteTimeIntegrator_PrevRese = 2;
  localDW->DiscreteTimeIntegrator_IC_LOADI = 1U;
}

/*
 * Output and update for atomic system:
 *    '<S6>/TOF'
 *    '<S6>/TOF1'
 *    '<S6>/TOF2'
 *    '<S425>/TOF'
 *    '<S427>/TOF1'
 *    '<S427>/TOF3'
 *    '<S667>/TOF'
 *    '<S831>/TOF'
 */
void Gen2_ref_TOF(boolean_T rtu_IN, real_T rtu_PT, rtB_TOF_Gen2_ref *localB,
                  rtDW_TOF_Gen2_ref *localDW, struct Gen2* inst)
{
  real_T rtb_Switch_aro;

  /* Switch: '<S329>/Switch' incorporates:
   *  Constant: '<S329>/Constant1'
   */
  if (rtu_IN) {
    rtb_Switch_aro = 0.0;
  } else {
    rtb_Switch_aro = rtu_PT;
  }

  /* End of Switch: '<S329>/Switch' */

  /* DiscreteIntegrator: '<S329>/Discrete-Time Integrator' */
  if (localDW->DiscreteTimeIntegrator_IC_LOADI != 0) {
    localDW->DiscreteTimeIntegrator_DSTATE = rtb_Switch_aro;
  }

  if (rtu_IN && (localDW->DiscreteTimeIntegrator_PrevRese <= 0)) {
    localDW->DiscreteTimeIntegrator_DSTATE = rtb_Switch_aro;
  }

  /* Logic: '<S329>/Logical Operator1' incorporates:
   *  DiscreteIntegrator: '<S329>/Discrete-Time Integrator'
   *  RelationalOperator: '<S329>/Relational Operator'
   */
  localB->LogicalOperator1 = !(localDW->DiscreteTimeIntegrator_DSTATE >= rtu_PT);

  /* Update for DiscreteIntegrator: '<S329>/Discrete-Time Integrator' incorporates:
   *  DataTypeConversion: '<S333>/Conversion'
   *  Logic: '<S329>/Logical Operator5'
   */
  localDW->DiscreteTimeIntegrator_IC_LOADI = 0U;
  localDW->DiscreteTimeIntegrator_DSTATE += 0.01 * (real_T)!rtu_IN;
  localDW->DiscreteTimeIntegrator_PrevRese = (int8_T)rtu_IN;
}

/*
 * Output and update for atomic system:
 *    '<S373>/2-point interpolation, with extrapolation'
 *    '<S373>/2-point interpolation, with extrapolation1'
 *    '<S473>/2-point interpolation, with extrapolation'
 *    '<S473>/2-point interpolation, with extrapolation1'
 *    '<S789>/2-point interpolation, with extrapolation'
 *    '<S789>/2-point interpolation, with extrapolation1'
 */
void upointinterpolationwithextrapol(real_T rtu_x, const real_T rtu_xDat[2],
  const real_T rtu_yDat[2], rtB_upointinterpolationwithextr *localB, struct Gen2* inst)
{
  real_T delta_x;
  delta_x = rtu_xDat[1] - rtu_xDat[0];
  if (fabs(delta_x) > 1.0E-7) {
    localB->y = (rtu_x - rtu_xDat[0]) / delta_x * (rtu_yDat[1] - rtu_yDat[0]) +
      rtu_yDat[0];
  } else {
    localB->y = (rtu_yDat[0] + rtu_yDat[1]) * 0.5;
  }
}

/*
 * Output and update for atomic system:
 *    '<S379>/MATLAB Function'
 *    '<S389>/MATLAB Function'
 */
void Gen2_ref_MATLABFunction_g(boolean_T rtu_reset, real_T rtu_u0, boolean_T
  rtu_LvrtFlg, real_T rtu_Y0Lvrt, rtB_MATLABFunction_Gen2_ref_k *localB,
  rtDW_MATLABFunction_Gen2_ref_f *localDW, struct Gen2* inst)
{
  if (!localDW->Y0OutTemp_not_empty) {
    localDW->Y0OutTemp = rtu_u0;
    localDW->Y0OutTemp_not_empty = true;
  }

  if (rtu_reset) {
    localB->ireset = true;
    localDW->Y0OutTemp = rtu_u0;
  } else if (rtu_LvrtFlg) {
    localB->ireset = true;
    localDW->Y0OutTemp = rtu_Y0Lvrt;
  } else {
    localB->ireset = false;
  }

  localB->Y0Out = localDW->Y0OutTemp;
}

/*
 * Output and update for atomic system:
 *    '<S379>/MATLAB Function1'
 *    '<S389>/MATLAB Function1'
 */
void Gen2_ref_MATLABFunction1(real_T rtu_LamIn, boolean_T rtu_LvrtFlg,
  rtB_MATLABFunction1_Gen2_ref *localB, rtDW_MATLABFunction1_Gen2_ref *localDW, struct Gen2* inst)
{
  if (!localDW->LamFix_not_empty) {
    localDW->LamFix = rtu_LamIn;
    localDW->LamFix_not_empty = true;
  }

  if (!rtu_LvrtFlg) {
    localB->LamOut = rtu_LamIn;
    localDW->LamFix = rtu_LamIn;
  } else {
    localB->LamOut = localDW->LamFix;
  }
}

/*
 * System initialize for atomic system:
 *    '<S344>/Pd_filt'
 *    '<S8>/Filter'
 *    '<S637>/Filter'
 *    '<S761>/Filter'
 *    '<S14>/Filter'
 *    '<S875>/Pd_filt'
 */
void Gen2_ref_Pd_filt_Init(rtDW_Pd_filt_Gen2_ref *localDW, struct Gen2* inst)
{
  /* InitializeConditions for DiscreteIntegrator: '<S396>/Discrete-Time Integrator' */
  localDW->DiscreteTimeIntegrator_IC_LOADI = 1U;
}

/*
 * Output and update for atomic system:
 *    '<S344>/Pd_filt'
 *    '<S8>/Filter'
 *    '<S637>/Filter'
 *    '<S761>/Filter'
 *    '<S14>/Filter'
 *    '<S875>/Pd_filt'
 */
void Gen2_ref_Pd_filt(real_T rtu_in, real_T rtu_T_filt, real_T rtu_x0, boolean_T
                      rtu_reset, rtB_Pd_filt_Gen2_ref *localB,
                      rtDW_Pd_filt_Gen2_ref *localDW, struct Gen2* inst)
{
  real_T tmp;
  boolean_T rtb_LogicalOperator_f;
  boolean_T rtb_RelationalOperator_py;

  /* RelationalOperator: '<S396>/Relational Operator' incorporates:
   *  Constant: '<S396>/Constant'
   */
  rtb_RelationalOperator_py = (rtu_T_filt > 0.0);

  /* Logic: '<S396>/Logical Operator' incorporates:
   *  Logic: '<S396>/Logical Operator1'
   */
  rtb_LogicalOperator_f = (rtu_reset || (!rtb_RelationalOperator_py));

  /* DiscreteIntegrator: '<S396>/Discrete-Time Integrator' */
  if (localDW->DiscreteTimeIntegrator_IC_LOADI != 0) {
    localDW->DiscreteTimeIntegrator_DSTATE = rtu_x0;
  }

  if (rtb_LogicalOperator_f || (localDW->DiscreteTimeIntegrator_PrevRese != 0))
  {
    localDW->DiscreteTimeIntegrator_DSTATE = rtu_x0;
  }

  /* Switch: '<S396>/Switch' */
  if (rtb_RelationalOperator_py) {
    /* Switch: '<S396>/Switch' incorporates:
     *  DiscreteIntegrator: '<S396>/Discrete-Time Integrator'
     */
    localB->Switch = localDW->DiscreteTimeIntegrator_DSTATE;
  } else {
    /* Switch: '<S396>/Switch' */
    localB->Switch = rtu_in;
  }

  /* End of Switch: '<S396>/Switch' */

  /* Update for DiscreteIntegrator: '<S396>/Discrete-Time Integrator' */
  localDW->DiscreteTimeIntegrator_IC_LOADI = 0U;

  /* Switch: '<S405>/Switch' incorporates:
   *  Abs: '<S405>/Abs'
   *  Constant: '<S405>/Constant2'
   *  RelationalOperator: '<S405>/Relational Operator'
   */
  if (2.2204460492503131E-16 >= fabs(rtu_T_filt)) {
    tmp = 2.2204460492503131E-16;
  } else {
    tmp = rtu_T_filt;
  }

  /* End of Switch: '<S405>/Switch' */

  /* Update for DiscreteIntegrator: '<S396>/Discrete-Time Integrator' incorporates:
   *  Product: '<S396>/Divide4'
   *  Sum: '<S396>/Sum4'
   */
  localDW->DiscreteTimeIntegrator_DSTATE += (rtu_in -
    localDW->DiscreteTimeIntegrator_DSTATE) / tmp * 0.01;
  localDW->DiscreteTimeIntegrator_PrevRese = (int8_T)rtb_LogicalOperator_f;
}

/*
 * System initialize for atomic system:
 *    '<S426>/TP'
 *    '<S426>/TP1'
 *    '<S427>/TP'
 *    '<S608>/SkipPulseWaitTP'
 *    '<S667>/TP'
 *    '<S667>/TP1'
 *    '<S831>/TP'
 *    '<S831>/TP1'
 */
void Gen2_ref_TP_Init(rtDW_TP_Gen2_ref *localDW, struct Gen2* inst)
{
  /* InitializeConditions for UnitDelay: '<S492>/Unit Delay2' */
  localDW->UnitDelay2_DSTATE = true;
}

/*
 * Output and update for atomic system:
 *    '<S426>/TP'
 *    '<S426>/TP1'
 *    '<S427>/TP'
 *    '<S608>/SkipPulseWaitTP'
 *    '<S667>/TP'
 *    '<S667>/TP1'
 *    '<S831>/TP'
 *    '<S831>/TP1'
 */
void Gen2_ref_TP(boolean_T rtu_IN, real_T rtu_PT, rtB_TP_Gen2_ref *localB,
                 rtDW_TP_Gen2_ref *localDW, struct Gen2* inst)
{
  real_T rtb_Switch2_ne;
  real_T rtb_UkYk1_gdc;

  /* Product: '<S498>/delta rise limit' incorporates:
   *  SampleTimeMath: '<S498>/sample time'
   *
   * About '<S498>/sample time':
   *  y = K where K = ( w * Ts )
   */
  rtb_Switch2_ne = 0.01;

  /* Outputs for Enabled SubSystem: '<S492>/Enabled Subsystem' incorporates:
   *  EnablePort: '<S496>/Enable'
   */
  /* Logic: '<S492>/Logical Operator3' incorporates:
   *  Logic: '<S492>/Logical Operator2'
   *  UnitDelay: '<S492>/Unit Delay2'
   */
  if ((!rtu_IN) && localDW->UnitDelay2_DSTATE) {
    /* Merge: '<S492>/Merge' incorporates:
     *  Constant: '<S492>/Constant10'
     *  Inport: '<S496>/In1'
     */
    localB->Merge = 0.0;
  }

  /* End of Logic: '<S492>/Logical Operator3' */
  /* End of Outputs for SubSystem: '<S492>/Enabled Subsystem' */

  /* Outputs for Enabled SubSystem: '<S492>/Enabled Subsystem1' incorporates:
   *  EnablePort: '<S497>/Enable'
   */
  if (rtu_IN) {
    /* Merge: '<S492>/Merge' incorporates:
     *  Inport: '<S497>/In1'
     */
    localB->Merge = rtu_PT;
  }

  /* End of Outputs for SubSystem: '<S492>/Enabled Subsystem1' */

  /* Sum: '<S498>/Difference Inputs1' incorporates:
   *  UnitDelay: '<S498>/Delay Input2'
   */
  rtb_UkYk1_gdc = localB->Merge - localDW->DelayInput2_DSTATE;

  /* Switch: '<S499>/Switch2' incorporates:
   *  RelationalOperator: '<S499>/LowerRelop1'
   */
  if (!(rtb_UkYk1_gdc > 0.01)) {
    /* Product: '<S498>/delta fall limit' incorporates:
     *  Constant: '<S492>/Constant9'
     *  SampleTimeMath: '<S498>/sample time'
     *
     * About '<S498>/sample time':
     *  y = K where K = ( w * Ts )
     */
    rtb_Switch2_ne = -99.990000000000009;

    /* Switch: '<S499>/Switch' incorporates:
     *  RelationalOperator: '<S499>/UpperRelop'
     */
    if (!(rtb_UkYk1_gdc < -99.990000000000009)) {
      rtb_Switch2_ne = rtb_UkYk1_gdc;
    }

    /* End of Switch: '<S499>/Switch' */
  }

  /* End of Switch: '<S499>/Switch2' */

  /* Sum: '<S498>/Difference Inputs2' incorporates:
   *  UnitDelay: '<S498>/Delay Input2'
   */
  rtb_UkYk1_gdc = rtb_Switch2_ne + localDW->DelayInput2_DSTATE;

  /* Logic: '<S492>/Logical Operator1' incorporates:
   *  Constant: '<S495>/Constant'
   *  RelationalOperator: '<S492>/Relational Operator1'
   *  RelationalOperator: '<S495>/Compare'
   */
  localB->LogicalOperator1 = ((rtb_UkYk1_gdc > 0.0) && (rtb_UkYk1_gdc < rtu_PT));

  /* Update for UnitDelay: '<S492>/Unit Delay2' incorporates:
   *  RelationalOperator: '<S492>/Relational Operator3'
   */
  localDW->UnitDelay2_DSTATE = (rtb_UkYk1_gdc >= rtu_PT);

  /* Update for UnitDelay: '<S498>/Delay Input2' */
  localDW->DelayInput2_DSTATE = rtb_UkYk1_gdc;
}

/*
 * System initialize for atomic system:
 *    '<S427>/TOF'
 *    '<S427>/TOF2'
 */
void Gen2_ref_TOF_p_Init(rtDW_TOF_Gen2_ref_f *localDW, struct Gen2* inst)
{
  /* InitializeConditions for DiscreteIntegrator: '<S511>/Discrete-Time Integrator' */
  localDW->DiscreteTimeIntegrator_PrevRese = 2;
  localDW->DiscreteTimeIntegrator_IC_LOADI = 1U;
}

/*
 * Output and update for atomic system:
 *    '<S427>/TOF'
 *    '<S427>/TOF2'
 * Common block description:
 *   Off Delay Timer
 */
void Gen2_ref_TOF_c(boolean_T rtu_IN, real32_T rtu_PT, rtB_TOF_Gen2_ref_j
                    *localB, rtDW_TOF_Gen2_ref_f *localDW, struct Gen2* inst)
{
  real32_T rtb_Switch_kwg;

  /* Switch: '<S511>/Switch' incorporates:
   *  Constant: '<S511>/Constant1'
   */
  if (rtu_IN) {
    rtb_Switch_kwg = 0.0F;
  } else {
    rtb_Switch_kwg = rtu_PT;
  }

  /* End of Switch: '<S511>/Switch' */

  /* DiscreteIntegrator: '<S511>/Discrete-Time Integrator' */
  if (localDW->DiscreteTimeIntegrator_IC_LOADI != 0) {
    localDW->DiscreteTimeIntegrator_DSTATE = rtb_Switch_kwg;
  }

  if (rtu_IN && (localDW->DiscreteTimeIntegrator_PrevRese <= 0)) {
    localDW->DiscreteTimeIntegrator_DSTATE = rtb_Switch_kwg;
  }

  /* Logic: '<S511>/Logical Operator1' incorporates:
   *  DiscreteIntegrator: '<S511>/Discrete-Time Integrator'
   *  RelationalOperator: '<S511>/Relational Operator'
   */
  localB->LogicalOperator1 = !(localDW->DiscreteTimeIntegrator_DSTATE >= rtu_PT);

  /* Update for DiscreteIntegrator: '<S511>/Discrete-Time Integrator' incorporates:
   *  DataTypeConversion: '<S529>/Conversion'
   *  Logic: '<S511>/Logical Operator5'
   */
  localDW->DiscreteTimeIntegrator_IC_LOADI = 0U;
  localDW->DiscreteTimeIntegrator_DSTATE += 0.01F * (real32_T)!rtu_IN;
  localDW->DiscreteTimeIntegrator_PrevRese = (int8_T)rtu_IN;
}

/*
 * System initialize for atomic system:
 *    '<S427>/TP_ActSat_CBV'
 *    '<S427>/TP_ActSat_TV'
 *    '<S427>/TP_Ign retard'
 *    '<S427>/TP_Misfire_OFF'
 *    '<S427>/TP_Misfire_OFF1'
 *    '<S427>/TP_Misfire_OFF2'
 *    '<S427>/TP_Misfire_ON'
 *    '<S427>/TP_Misfire_ON_2nd time'
 */
void Gen2_ref_TP_ActSat_CBV_Init(rtDW_TP_ActSat_CBV_Gen2_ref *localDW, struct Gen2* inst)
{
  /* InitializeConditions for UnitDelay: '<S516>/Unit Delay2' */
  localDW->UnitDelay2_DSTATE = true;
}

/*
 * Output and update for atomic system:
 *    '<S427>/TP_ActSat_CBV'
 *    '<S427>/TP_ActSat_TV'
 *    '<S427>/TP_Ign retard'
 *    '<S427>/TP_Misfire_OFF'
 *    '<S427>/TP_Misfire_OFF1'
 *    '<S427>/TP_Misfire_OFF2'
 *    '<S427>/TP_Misfire_ON'
 *    '<S427>/TP_Misfire_ON_2nd time'
 */
void Gen2_ref_TP_ActSat_CBV(boolean_T rtu_IN, real_T rtu_PT,
  rtB_TP_ActSat_CBV_Gen2_ref *localB, rtDW_TP_ActSat_CBV_Gen2_ref *localDW, struct Gen2* inst)
{
  real_T rtb_Switch2_fj;
  real_T rtb_UkYk1_d;

  /* Product: '<S541>/delta rise limit' incorporates:
   *  SampleTimeMath: '<S541>/sample time'
   *
   * About '<S541>/sample time':
   *  y = K where K = ( w * Ts )
   */
  rtb_Switch2_fj = 0.01;

  /* Outputs for Enabled SubSystem: '<S516>/Enabled Subsystem' incorporates:
   *  EnablePort: '<S539>/Enable'
   */
  /* Logic: '<S516>/Logical Operator3' incorporates:
   *  Logic: '<S516>/Logical Operator2'
   *  UnitDelay: '<S516>/Unit Delay2'
   */
  if ((!rtu_IN) && localDW->UnitDelay2_DSTATE) {
    /* Merge: '<S516>/Merge' incorporates:
     *  Constant: '<S516>/Constant10'
     *  Inport: '<S539>/In1'
     */
    localB->Merge = 0.0;
  }

  /* End of Logic: '<S516>/Logical Operator3' */
  /* End of Outputs for SubSystem: '<S516>/Enabled Subsystem' */

  /* Outputs for Enabled SubSystem: '<S516>/Enabled Subsystem1' incorporates:
   *  EnablePort: '<S540>/Enable'
   */
  if (rtu_IN) {
    /* Merge: '<S516>/Merge' incorporates:
     *  Inport: '<S540>/In1'
     */
    localB->Merge = rtu_PT;
  }

  /* End of Outputs for SubSystem: '<S516>/Enabled Subsystem1' */

  /* Sum: '<S541>/Difference Inputs1' incorporates:
   *  UnitDelay: '<S541>/Delay Input2'
   */
  rtb_UkYk1_d = localB->Merge - localDW->DelayInput2_DSTATE;

  /* Switch: '<S542>/Switch2' incorporates:
   *  RelationalOperator: '<S542>/LowerRelop1'
   */
  if (!(rtb_UkYk1_d > 0.01)) {
    /* Product: '<S541>/delta fall limit' incorporates:
     *  Constant: '<S516>/Constant9'
     *  SampleTimeMath: '<S541>/sample time'
     *
     * About '<S541>/sample time':
     *  y = K where K = ( w * Ts )
     */
    rtb_Switch2_fj = -99.990000000000009;

    /* Switch: '<S542>/Switch' incorporates:
     *  RelationalOperator: '<S542>/UpperRelop'
     */
    if (!(rtb_UkYk1_d < -99.990000000000009)) {
      rtb_Switch2_fj = rtb_UkYk1_d;
    }

    /* End of Switch: '<S542>/Switch' */
  }

  /* End of Switch: '<S542>/Switch2' */

  /* Sum: '<S541>/Difference Inputs2' incorporates:
   *  UnitDelay: '<S541>/Delay Input2'
   */
  rtb_UkYk1_d = rtb_Switch2_fj + localDW->DelayInput2_DSTATE;

  /* Logic: '<S516>/Logical Operator1' incorporates:
   *  Constant: '<S538>/Constant'
   *  RelationalOperator: '<S516>/Relational Operator1'
   *  RelationalOperator: '<S538>/Compare'
   */
  localB->LogicalOperator1 = ((rtb_UkYk1_d > 0.0) && (rtb_UkYk1_d < rtu_PT));

  /* Update for UnitDelay: '<S516>/Unit Delay2' incorporates:
   *  RelationalOperator: '<S516>/Relational Operator3'
   */
  localDW->UnitDelay2_DSTATE = (rtb_UkYk1_d >= rtu_PT);

  /* Update for UnitDelay: '<S541>/Delay Input2' */
  localDW->DelayInput2_DSTATE = rtb_UkYk1_d;
}

/*
 * Output and update for atomic system:
 *    '<S589>/MATLAB Function'
 *    '<S582>/MATLAB Function'
 *    '<S582>/MATLAB Function1'
 *    '<S633>/MATLAB Function'
 *    '<S19>/MATLAB Function'
 */
void Gen2_ref_MATLABFunction_n(real_T rtu_u, real_T rtu_eps,
  rtB_MATLABFunction_Gen2_ref_o *localB, rtDW_MATLABFunction_Gen2_ref_k *localDW, struct Gen2* inst)
{
  real_T delta;
  delta = rtu_u - localDW->y_z;
  if (delta > rtu_eps) {
    localB->y = localDW->y_z + 1.0;
  } else if (delta < -rtu_eps) {
    localB->y = localDW->y_z - 1.0;
  } else {
    localB->y = localDW->y_z;
  }

  localDW->y_z = localB->y;
}

/*
 * System initialize for atomic system:
 *    '<S630>/Filter'
 *    '<S636>/Filter'
 */
void Gen2_ref_Filter_Init(rtDW_Filter_Gen2_ref *localDW, struct Gen2* inst)
{
  /* InitializeConditions for DiscreteIntegrator: '<S665>/Discrete-Time Integrator' */
  localDW->DiscreteTimeIntegrator_IC_LOADI = 1U;
}

/*
 * Output and update for atomic system:
 *    '<S630>/Filter'
 *    '<S636>/Filter'
 */
void Gen2_ref_Filter(real_T rtu_in, real_T rtu_x0, boolean_T rtu_reset,
                     rtB_Filter_Gen2_ref *localB, const rtC_Filter_Gen2_ref
                     *localC, rtDW_Filter_Gen2_ref *localDW, struct Gen2* inst)
{
  boolean_T rtb_LogicalOperator_g1;

  /* Logic: '<S665>/Logical Operator' */
  rtb_LogicalOperator_g1 = (rtu_reset || localC->LogicalOperator1);

  /* DiscreteIntegrator: '<S665>/Discrete-Time Integrator' */
  if (localDW->DiscreteTimeIntegrator_IC_LOADI != 0) {
    localDW->DiscreteTimeIntegrator_DSTATE = rtu_x0;
  }

  if (rtb_LogicalOperator_g1 || (localDW->DiscreteTimeIntegrator_PrevRese != 0))
  {
    localDW->DiscreteTimeIntegrator_DSTATE = rtu_x0;
  }

  /* Switch: '<S665>/Switch' */
  if (localC->RelationalOperator_g) {
    /* Switch: '<S665>/Switch' incorporates:
     *  DiscreteIntegrator: '<S665>/Discrete-Time Integrator'
     */
    localB->Switch = localDW->DiscreteTimeIntegrator_DSTATE;
  } else {
    /* Switch: '<S665>/Switch' */
    localB->Switch = rtu_in;
  }

  /* End of Switch: '<S665>/Switch' */

  /* Update for DiscreteIntegrator: '<S665>/Discrete-Time Integrator' incorporates:
   *  Product: '<S665>/Divide4'
   *  Sum: '<S665>/Sum4'
   */
  localDW->DiscreteTimeIntegrator_IC_LOADI = 0U;
  localDW->DiscreteTimeIntegrator_DSTATE += (rtu_in -
    localDW->DiscreteTimeIntegrator_DSTATE) / localC->Switch * 0.01;
  localDW->DiscreteTimeIntegrator_PrevRese = (int8_T)rtb_LogicalOperator_g1;
}

/*
 * Output and update for atomic system:
 *    '<S666>/Ke Map Update'
 *    '<S830>/Ke Map Update'
 */
void Gen2_ref_KeMapUpdate(real_T rtu_in, boolean_T rtu_reset, real_T rtu_Ke_map,
  boolean_T rtu_resetTrans, boolean_T rtu_resetTrans_f, const tGen2Parameter
  *rtu_para, rtB_KeMapUpdate_Gen2_ref *localB, rtDW_KeMapUpdate_Gen2_ref
  *localDW, struct Gen2* inst)
{
  real_T rtb_RelationalOperator_gj;
  real_T rtb_Switch_cs;
  real_T rtb_Switch_mvl;
  boolean_T rtb_LogicalOperator_lv;
  boolean_T rtb_RelationalOperator_kzb;

  /* Sum: '<S671>/Sum' incorporates:
   *  Product: '<S671>/Divide2'
   */
  rtb_Switch_mvl = rtu_para->SpeedCtrl.rTiF_KeEstIncrAfterTrans * (real_T)
    rtu_resetTrans + rtu_para->SpeedCtrl.rTiF_KeEstDiffMapUpdate;

  /* RelationalOperator: '<S671>/Relational Operator' incorporates:
   *  Constant: '<S671>/Constant'
   */
  rtb_RelationalOperator_kzb = (rtb_Switch_mvl > 0.0);

  /* Logic: '<S671>/Logical Operator' incorporates:
   *  Logic: '<S671>/Logical Operator1'
   */
  rtb_LogicalOperator_lv = (rtu_reset || rtu_resetTrans_f ||
    (!rtb_RelationalOperator_kzb));

  /* DiscreteIntegrator: '<S671>/Discrete-Time Integrator' */
  if (rtb_LogicalOperator_lv || (localDW->DiscreteTimeIntegrator_PrevRese != 0))
  {
    localDW->DiscreteTimeIntegrator_DSTATE = 0.0;
  }

  /* Sum: '<S671>/Sum3' */
  rtb_Switch_cs = rtu_in - rtu_Ke_map;

  /* Switch: '<S671>/Switch' incorporates:
   *  DiscreteIntegrator: '<S671>/Discrete-Time Integrator'
   */
  if (rtb_RelationalOperator_kzb) {
    rtb_RelationalOperator_gj = localDW->DiscreteTimeIntegrator_DSTATE;
  } else {
    rtb_RelationalOperator_gj = rtb_Switch_cs;
  }

  /* End of Switch: '<S671>/Switch' */

  /* Sum: '<S671>/Sum1' */
  localB->Sum1 = rtb_RelationalOperator_gj + rtu_Ke_map;

  /* Switch: '<S674>/Switch' incorporates:
   *  Abs: '<S674>/Abs'
   *  Constant: '<S674>/Constant2'
   *  RelationalOperator: '<S674>/Relational Operator'
   */
  if (2.2204460492503131E-16 >= fabs(rtb_Switch_mvl)) {
    rtb_Switch_mvl = 2.2204460492503131E-16;
  }

  /* End of Switch: '<S674>/Switch' */

  /* Update for DiscreteIntegrator: '<S671>/Discrete-Time Integrator' incorporates:
   *  Product: '<S671>/Divide4'
   *  Sum: '<S671>/Sum4'
   */
  localDW->DiscreteTimeIntegrator_DSTATE += (rtb_Switch_cs -
    localDW->DiscreteTimeIntegrator_DSTATE) / rtb_Switch_mvl * 0.01;
  localDW->DiscreteTimeIntegrator_PrevRese = (int8_T)rtb_LogicalOperator_lv;
}

/* Function for MATLAB Function: '<S666>/MATLAB Function1' */
static real_T Gen2_ref_maximum(const real_T x[13], struct Gen2* inst)
{
  real_T ex;
  int32_T idx;
  int32_T k;
  boolean_T exitg1;
  if (!rtIsNaN(x[0])) {
    idx = 1;
  } else {
    idx = 0;
    k = 2;
    exitg1 = false;
    while ((!exitg1) && (k < 14)) {
      if (!rtIsNaN(x[k - 1])) {
        idx = k;
        exitg1 = true;
      } else {
        k++;
      }
    }
  }

  if (idx == 0) {
    ex = x[0];
  } else {
    ex = x[idx - 1];
    while (idx + 1 <= 13) {
      if (ex < x[idx]) {
        ex = x[idx];
      }

      idx++;
    }
  }

  return ex;
}

/*
 * Output and update for atomic system:
 *    '<S666>/MATLAB Function1'
 *    '<S830>/MATLAB Function1'
 */
void Gen2_ref_MATLABFunction1_m(const real_T rtu_x_ref[13], const real_T
  rtu_y_ref[13], real_T rtu_epsilon, real_T rtu_x_f, real_T rtu_y_act, boolean_T
  rtu_reset, boolean_T rtu_issteady, rtB_MATLABFunction1_Gen2_ref_h *localB,
  rtDW_MATLABFunction1_Gen2_ref_c *localDW, struct Gen2* inst)
{
  real_T delta_y;
  real_T delta_y_tmp_tmp;
  real_T delta_y_tmp_tmp_0;
  real_T u0;
  real_T x;
  real_T y_map_tmp;
  int32_T i;
  int32_T k;
  boolean_T exitg1;
  if ((!localDW->y_map_not_empty) || rtu_reset) {
    localDW->y_map_not_empty = true;
    for (i = 0; i < 13; i++) {
      localDW->y_map[i] = rtu_y_ref[i];
      localDW->x_map[i] = rtu_x_ref[i];
    }
  }

  if (Gen2_ref_maximum(localDW->y_map, inst) < 0.1) {
    for (i = 0; i < 13; i++) {
      localDW->y_map[i] = rtu_y_ref[i];
    }
  }

  if (!rtIsNaN(localDW->x_map[0])) {
    i = 1;
  } else {
    i = 0;
    k = 2;
    exitg1 = false;
    while ((!exitg1) && (k < 14)) {
      if (!rtIsNaN(localDW->x_map[k - 1])) {
        i = k;
        exitg1 = true;
      } else {
        k++;
      }
    }
  }

  if (i == 0) {
    x = localDW->x_map[0];
  } else {
    x = localDW->x_map[i - 1];
    while (i + 1 <= 13) {
      if (x > localDW->x_map[i]) {
        x = localDW->x_map[i];
      }

      i++;
    }
  }

  if ((!(x >= rtu_x_f)) && (!rtIsNaN(rtu_x_f))) {
    x = rtu_x_f;
  }

  u0 = Gen2_ref_maximum(localDW->x_map, inst);
  if ((u0 <= x) || rtIsNaN(x)) {
    x = u0;
  }

  k = 0;
  if (!(x < localDW->x_map[0])) {
    for (i = 0; i < 13; i++) {
      if (x > localDW->x_map[i]) {
        k = i;
      }
    }
  }

  if (k + 1 < 13) {
    if (rtu_issteady && (!rtu_reset)) {
      u0 = localDW->y_map[k + 1];
      delta_y_tmp_tmp = x - localDW->x_map[k];
      delta_y_tmp_tmp_0 = localDW->x_map[k + 1];
      delta_y = delta_y_tmp_tmp / (delta_y_tmp_tmp_0 - localDW->x_map[k]) * (u0
        - localDW->y_map[k]) + localDW->y_map[k];
      delta_y = ((1.0 - rtu_epsilon) * delta_y + rtu_epsilon * rtu_y_act) -
        delta_y;
      x = delta_y_tmp_tmp_0 - x;
      delta_y_tmp_tmp_0 = delta_y_tmp_tmp + x;
      y_map_tmp = delta_y_tmp_tmp_0 * x;
      x = (delta_y_tmp_tmp * delta_y_tmp_tmp + y_map_tmp) - delta_y_tmp_tmp * x;
      localDW->y_map[k] += y_map_tmp * delta_y / x;
      localDW->y_map[k + 1] = delta_y_tmp_tmp_0 * delta_y_tmp_tmp * delta_y / x
        + u0;
    }
  } else if (rtu_issteady && (!rtu_reset)) {
    localDW->y_map[12] = (1.0 - rtu_epsilon) * localDW->y_map[12] + rtu_epsilon *
      rtu_y_act;
  }

  for (i = 0; i < 13; i++) {
    localB->y_map_new[i] = localDW->y_map[i];
  }
}

real_T rt_roundd_snf(real_T u, struct Gen2* inst)
{
  real_T y;
  if (fabs(u) < 4.503599627370496E+15) {
    if (u >= 0.5) {
      y = floor(u + 0.5);
    } else if (u > -0.5) {
      y = u * 0.0;
    } else {
      y = ceil(u - 0.5);
    }
  } else {
    y = u;
  }

  return y;
}

real_T rt_powd_snf(real_T u0, real_T u1, struct Gen2* inst)
{
  real_T tmp;
  real_T tmp_0;
  real_T y;
  if (rtIsNaN(u0) || rtIsNaN(u1)) {
    y = (rtNaN);
  } else {
    tmp = fabs(u0);
    tmp_0 = fabs(u1);
    if (rtIsInf(u1)) {
      if (tmp == 1.0) {
        y = 1.0;
      } else if (tmp > 1.0) {
        if (u1 > 0.0) {
          y = (rtInf);
        } else {
          y = 0.0;
        }
      } else if (u1 > 0.0) {
        y = 0.0;
      } else {
        y = (rtInf);
      }
    } else if (tmp_0 == 0.0) {
      y = 1.0;
    } else if (tmp_0 == 1.0) {
      if (u1 > 0.0) {
        y = u0;
      } else {
        y = 1.0 / u0;
      }
    } else if (u1 == 2.0) {
      y = u0 * u0;
    } else if ((u1 == 0.5) && (u0 >= 0.0)) {
      y = sqrt(u0);
    } else if ((u0 < 0.0) && (u1 > floor(u1))) {
      y = (rtNaN);
    } else {
      y = pow(u0, u1);
    }
  }

  return y;
}

/* Function for MATLAB Function: '<S716>/MATLAB Function' */
static real_T Gen2_ref_minimum(const real_T x[13], struct Gen2* inst)
{
  real_T ex;
  int32_T idx;
  int32_T k;
  boolean_T exitg1;
  if (!rtIsNaN(x[0])) {
    idx = 1;
  } else {
    idx = 0;
    k = 2;
    exitg1 = false;
    while ((!exitg1) && (k < 14)) {
      if (!rtIsNaN(x[k - 1])) {
        idx = k;
        exitg1 = true;
      } else {
        k++;
      }
    }
  }

  if (idx == 0) {
    ex = x[0];
  } else {
    ex = x[idx - 1];
    while (idx + 1 <= 13) {
      if (ex > x[idx]) {
        ex = x[idx];
      }

      idx++;
    }
  }

  return ex;
}

/* Function for MATLAB Function: '<S714>/MATLAB Function1' */
static real_T Gen2_ref_maximum_f(const real_T x[13], struct Gen2* inst)
{
  real_T ex;
  int32_T idx;
  int32_T k;
  boolean_T exitg1;
  if (!rtIsNaN(x[0])) {
    idx = 1;
  } else {
    idx = 0;
    k = 2;
    exitg1 = false;
    while ((!exitg1) && (k < 14)) {
      if (!rtIsNaN(x[k - 1])) {
        idx = k;
        exitg1 = true;
      } else {
        k++;
      }
    }
  }

  if (idx == 0) {
    ex = x[0];
  } else {
    ex = x[idx - 1];
    while (idx + 1 <= 13) {
      if (ex < x[idx]) {
        ex = x[idx];
      }

      idx++;
    }
  }

  return ex;
}

/* Function for MATLAB Function: '<S431>/LQR Controller 3states' */
static void Gen2_ref_diag(const real_T v[2], real_T d[4], struct Gen2* inst)
{
  d[1] = 0.0;
  d[2] = 0.0;
  d[0] = v[0];
  d[3] = v[1];
}

/* Function for MATLAB Function: '<S431>/LQR Controller 3states' */
static void Gen2_ref_diag_i(const real_T v[4], real_T d[16], struct Gen2* inst)
{
  int32_T i;
  for (i = 0; i < 16; i++) {
    d[i] = 0.0;
  }

  d[0] = v[0];
  d[5] = v[1];
  d[10] = v[2];
  d[15] = v[3];
}

/* Function for MATLAB Function: '<S431>/LQR Controller 3states' */
static void Gen2_ref_diag_i2(const real_T v[3], real_T d[9], struct Gen2* inst)
{
  int32_T i;
  for (i = 0; i < 9; i++) {
    d[i] = 0.0;
  }

  d[0] = v[0];
  d[4] = v[1];
  d[8] = v[2];
}

/* Function for MATLAB Function: '<S431>/LQR Controller 3states' */
static void Gen2_ref_state_space_d(const real_T x[3], const real_T p[22], real_T
  Ke_in, real_T Phi[9], real_T h[12], real_T hd[3], struct Gen2* inst)
{
  real_T Phi_tmp;
  real_T Phi_tmp_0;
  real_T Phi_tmp_1;
  real_T a_tmp;
  a_tmp = x[2] * p[8] + 1.0;
  Phi[0] = 1.0;
  Phi_tmp = a_tmp * p[3];
  Phi[3] = Ke_in * p[2] / Phi_tmp;
  Phi[6] = -(Ke_in * p[8] * p[2] * x[1]) / (a_tmp * a_tmp * p[3]);
  Phi[1] = 0.0;
  Phi_tmp_0 = p[2] / p[5];
  Phi[4] = 1.0 - Phi_tmp_0;
  Phi[7] = 0.0;
  Phi[2] = 0.0;
  Phi[5] = 0.0;
  Phi_tmp_1 = p[2] / p[6];
  Phi[8] = 1.0 - Phi_tmp_1;
  h[0] = 0.0;
  h[3] = 0.0;
  h[6] = p[7] * Ke_in * p[2] * x[1] / Phi_tmp;
  h[9] = -(p[11] * Ke_in * p[2] * x[1]) / ((p[12] - p[11] * p[16]) * p[3] *
    a_tmp);
  h[1] = Phi_tmp_0;
  h[4] = 0.0;
  h[7] = 0.0;
  h[10] = 0.0;
  h[2] = 0.0;
  h[5] = Phi_tmp_1;
  h[8] = 0.0;
  h[11] = 0.0;
  hd[0] = -p[2] / p[3];
  hd[1] = 0.0;
  hd[2] = 0.0;
}

/* Function for MATLAB Function: '<S431>/LQR Controller 3states' */
static void Gen2_ref_diag_i2a(const real_T v[6], real_T d[36], struct Gen2* inst)
{
  int32_T j;
  for (j = 0; j < 36; j++) {
    d[j] = 0.0;
  }

  for (j = 0; j < 6; j++) {
    d[j + 6 * j] = v[j];
  }
}

/* Function for MATLAB Function: '<S431>/LQR Controller 3states' */
static real_T Gen2_ref_det(const real_T x[9], struct Gen2* inst)
{
  real_T A[9];
  real_T s;
  real_T smax;
  real_T y;
  int32_T c;
  int32_T c_ix;
  int32_T c_k;
  int32_T ijA;
  int32_T ix;
  int32_T iy;
  int32_T j;
  int32_T jj;
  int8_T ipiv[3];
  boolean_T isodd;
  for (j = 0; j < 9; j++) {
    A[j] = x[j];
  }

  ipiv[0] = 1;
  ipiv[1] = 2;
  for (j = 0; j < 2; j++) {
    jj = j << 2;
    iy = 0;
    ix = jj;
    smax = fabs(A[jj]);
    for (c_k = 2; c_k <= 3 - j; c_k++) {
      ix++;
      s = fabs(A[ix]);
      if (s > smax) {
        iy = c_k - 1;
        smax = s;
      }
    }

    if (A[jj + iy] != 0.0) {
      if (iy != 0) {
        iy += j;
        ipiv[j] = (int8_T)(iy + 1);
        smax = A[j];
        A[j] = A[iy];
        A[iy] = smax;
        smax = A[j + 3];
        A[j + 3] = A[iy + 3];
        A[iy + 3] = smax;
        smax = A[j + 6];
        A[j + 6] = A[iy + 6];
        A[iy + 6] = smax;
      }

      iy = (jj - j) + 3;
      for (ix = jj + 1; ix < iy; ix++) {
        A[ix] /= A[jj];
      }
    }

    iy = jj;
    ix = jj + 3;
    for (c_k = 0; c_k <= 1 - j; c_k++) {
      if (A[ix] != 0.0) {
        smax = -A[ix];
        c_ix = jj + 1;
        ijA = iy + 4;
        c = (iy - j) + 6;
        while (ijA + 1 <= c) {
          A[ijA] += A[c_ix] * smax;
          c_ix++;
          ijA++;
        }
      }

      ix += 3;
      iy += 3;
    }
  }

  isodd = (ipiv[0] > 1);
  y = A[0] * A[4] * A[8];
  if (ipiv[1] > 2) {
    isodd = !isodd;
  }

  if (isodd) {
    y = -y;
  }

  return y;
}

/* Function for MATLAB Function: '<S431>/LQR Controller 3states' */
static void Gen2_ref_mrdiv(const real_T A[18], const real_T B[9], real_T Y[18], struct Gen2* inst)
{
  real_T b_A[9];
  real_T a21;
  real_T maxval;
  int32_T Y_tmp;
  int32_T Y_tmp_0;
  int32_T Y_tmp_1;
  int32_T r1;
  int32_T r2;
  int32_T r3;
  int32_T rtemp;
  for (r1 = 0; r1 < 9; r1++) {
    b_A[r1] = B[r1];
  }

  r1 = 0;
  r2 = 1;
  r3 = 2;
  maxval = fabs(B[0]);
  a21 = fabs(B[1]);
  if (a21 > maxval) {
    maxval = a21;
    r1 = 1;
    r2 = 0;
  }

  if (fabs(B[2]) > maxval) {
    r1 = 2;
    r2 = 1;
    r3 = 0;
  }

  b_A[r2] = B[r2] / B[r1];
  b_A[r3] /= b_A[r1];
  b_A[r2 + 3] -= b_A[r1 + 3] * b_A[r2];
  b_A[r3 + 3] -= b_A[r1 + 3] * b_A[r3];
  b_A[r2 + 6] -= b_A[r1 + 6] * b_A[r2];
  b_A[r3 + 6] -= b_A[r1 + 6] * b_A[r3];
  if (fabs(b_A[r3 + 3]) > fabs(b_A[r2 + 3])) {
    rtemp = r2;
    r2 = r3;
    r3 = rtemp;
  }

  b_A[r3 + 3] /= b_A[r2 + 3];
  b_A[r3 + 6] -= b_A[r3 + 3] * b_A[r2 + 6];
  for (rtemp = 0; rtemp < 6; rtemp++) {
    Y_tmp = 6 * r1 + rtemp;
    Y[Y_tmp] = A[rtemp] / b_A[r1];
    Y_tmp_0 = 6 * r2 + rtemp;
    Y[Y_tmp_0] = A[rtemp + 6] - b_A[r1 + 3] * Y[Y_tmp];
    Y_tmp_1 = 6 * r3 + rtemp;
    Y[Y_tmp_1] = A[rtemp + 12] - b_A[r1 + 6] * Y[Y_tmp];
    Y[Y_tmp_0] /= b_A[r2 + 3];
    Y[Y_tmp_1] -= b_A[r2 + 6] * Y[Y_tmp_0];
    Y[Y_tmp_1] /= b_A[r3 + 6];
    Y[Y_tmp_0] -= b_A[r3 + 3] * Y[Y_tmp_1];
    Y[Y_tmp] -= Y[Y_tmp_1] * b_A[r3];
    Y[Y_tmp] -= Y[Y_tmp_0] * b_A[r2];
  }
}

/* Function for MATLAB Function: '<S431>/LQR Controller 3states' */
static void Gen2_ref_mldivide(const real_T A[16], const real_T B[12], real_T Y
  [12], struct Gen2* inst)
{
  real_T b_A[16];
  real_T s;
  real_T smax;
  int32_T b_j;
  int32_T c;
  int32_T c_ix;
  int32_T c_k;
  int32_T ijA;
  int32_T ix;
  int32_T iy;
  int32_T jj;
  int8_T ipiv[4];
  int8_T ipiv_0;
  for (b_j = 0; b_j < 16; b_j++) {
    b_A[b_j] = A[b_j];
  }

  for (b_j = 0; b_j < 12; b_j++) {
    Y[b_j] = B[b_j];
  }

  ipiv[0] = 1;
  ipiv[1] = 2;
  ipiv[2] = 3;
  ipiv[3] = 4;
  for (b_j = 0; b_j < 3; b_j++) {
    jj = b_j * 5;
    iy = 0;
    ix = jj;
    smax = fabs(b_A[jj]);
    for (c_k = 2; c_k <= 4 - b_j; c_k++) {
      ix++;
      s = fabs(b_A[ix]);
      if (s > smax) {
        iy = c_k - 1;
        smax = s;
      }
    }

    if (b_A[jj + iy] != 0.0) {
      if (iy != 0) {
        c_k = b_j + iy;
        ipiv[b_j] = (int8_T)(c_k + 1);
        smax = b_A[b_j];
        b_A[b_j] = b_A[c_k];
        b_A[c_k] = smax;
        smax = b_A[b_j + 4];
        b_A[b_j + 4] = b_A[c_k + 4];
        b_A[c_k + 4] = smax;
        smax = b_A[b_j + 8];
        b_A[b_j + 8] = b_A[c_k + 8];
        b_A[c_k + 8] = smax;
        smax = b_A[b_j + 12];
        b_A[b_j + 12] = b_A[c_k + 12];
        b_A[c_k + 12] = smax;
      }

      iy = (jj - b_j) + 4;
      for (ix = jj + 1; ix < iy; ix++) {
        b_A[ix] /= b_A[jj];
      }
    }

    iy = jj;
    ix = jj + 4;
    for (c_k = 0; c_k <= 2 - b_j; c_k++) {
      if (b_A[ix] != 0.0) {
        smax = -b_A[ix];
        c_ix = jj + 1;
        ijA = iy + 5;
        c = (iy - b_j) + 8;
        while (ijA + 1 <= c) {
          b_A[ijA] += b_A[c_ix] * smax;
          c_ix++;
          ijA++;
        }
      }

      ix += 4;
      iy += 4;
    }
  }

  for (b_j = 0; b_j < 3; b_j++) {
    ipiv_0 = ipiv[b_j];
    if (b_j + 1 != ipiv_0) {
      smax = Y[b_j];
      Y[b_j] = Y[ipiv_0 - 1];
      Y[ipiv_0 - 1] = smax;
      smax = Y[b_j + 4];
      Y[b_j + 4] = Y[ipiv_0 + 3];
      Y[ipiv_0 + 3] = smax;
      smax = Y[b_j + 8];
      Y[b_j + 8] = Y[ipiv_0 + 7];
      Y[ipiv_0 + 7] = smax;
    }
  }

  for (b_j = 0; b_j < 3; b_j++) {
    jj = b_j << 2;
    if (Y[jj] != 0.0) {
      for (c_k = 2; c_k < 5; c_k++) {
        iy = (c_k + jj) - 1;
        Y[iy] -= b_A[c_k - 1] * Y[jj];
      }
    }

    if (Y[jj + 1] != 0.0) {
      for (c_k = 3; c_k < 5; c_k++) {
        iy = (c_k + jj) - 1;
        Y[iy] -= Y[jj + 1] * b_A[c_k + 3];
      }
    }

    smax = Y[jj + 2];
    if (smax != 0.0) {
      Y[jj + 3] -= smax * b_A[11];
    }
  }

  for (b_j = 0; b_j < 3; b_j++) {
    jj = b_j << 2;
    smax = Y[jj + 3];
    if (smax != 0.0) {
      Y[jj + 3] = smax / b_A[15];
      for (c_k = 0; c_k < 3; c_k++) {
        iy = c_k + jj;
        Y[iy] -= Y[jj + 3] * b_A[c_k + 12];
      }
    }

    smax = Y[jj + 2];
    if (smax != 0.0) {
      Y[jj + 2] = smax / b_A[10];
      for (c_k = 0; c_k < 2; c_k++) {
        iy = c_k + jj;
        Y[iy] -= Y[jj + 2] * b_A[c_k + 8];
      }
    }

    smax = Y[jj + 1];
    if (smax != 0.0) {
      Y[jj + 1] = smax / b_A[5];
      Y[jj] -= Y[jj + 1] * b_A[4];
    }

    if (Y[jj] != 0.0) {
      Y[jj] /= b_A[0];
    }
  }
}

/* Function for MATLAB Function: '<S431>/LQR Controller 3states' */
static void Gen2_ref_integrate_model(real_T x0[3], const real_T K[12], const
  real_T u2_past[100], real_T d, const real_T x_disturb[3], const real_T Bd[9],
  real_T x_disturb1_map, const real_T u_sp[4], const real_T x_sp[3], int16_T N,
  const real_T u_min[4], const real_T u_max[4], const real_T p[22], struct Gen2* inst)
{
  real_T u_k[4];
  real_T u_k_0;
  real_T u_max_0;
  real_T u_min_0;
  real_T x_sp_idx_0;
  real_T x_sp_idx_1;
  real_T x_sp_idx_2;
  int32_T k;
  int32_T m;
  for (k = 0; k < N; k++) {
    x_sp_idx_0 = x_sp[0] - x0[0];
    x_sp_idx_1 = x_sp[1] - x0[1];
    x_sp_idx_2 = x_sp[2] - x0[2];
    for (m = 0; m < 4; m++) {
      u_min_0 = u_min[m];
      u_max_0 = u_max[m];
      u_k_0 = u_sp[m] - ((K[m + 4] * x_sp_idx_1 + K[m] * x_sp_idx_0) + K[m + 8] *
                         x_sp_idx_2);
      if (u_k_0 > u_max_0) {
        u_k_0 = u_max_0;
      } else if (u_k_0 < u_min_0) {
        u_k_0 = u_min_0;
      }

      u_k[m] = u_k_0;
    }

    x_sp_idx_0 = x0[1] * p[10] + p[9];
    x_sp_idx_1 = 1.0 / p[5] * (u_k[0] - x0[1]);
    x_sp_idx_2 = 1.0 / p[6] * (u2_past[k] - x0[2]);
    x0[0] += (((1.0 / (x0[2] * p[8] + 1.0) * p[4] * x0[1] * (u_k[2] * p[7] + 1.0)
                - d) * (1.0 / p[3]) + x_disturb[0] * Bd[0]) + x_disturb1_map *
              Bd[0]) * p[2];
    if ((x_sp_idx_0 <= x_sp_idx_1) || rtIsNaN(x_sp_idx_1)) {
      x_sp_idx_1 = x_sp_idx_0;
    }

    x0[1] += x_sp_idx_1 * p[2];
    x0[2] += x_sp_idx_2 * p[2];
  }
}

/* Function for MATLAB Function: '<S431>/LQR Controller 3states' */
static void Gen2_ref_mldivide_j(const real_T A[4], const real_T B[12], real_T Y
  [12], struct Gen2* inst)
{
  real_T Y_tmp_0;
  real_T a21;
  real_T a22;
  real_T a22_tmp;
  int32_T Y_tmp;
  int32_T k;
  int32_T r1;
  int32_T r2;
  if (fabs(A[1]) > fabs(A[0])) {
    r1 = 1;
    r2 = 0;
  } else {
    r1 = 0;
    r2 = 1;
  }

  a21 = A[r2] / A[r1];
  a22_tmp = A[r1 + 2];
  a22 = A[r2 + 2] - a22_tmp * a21;
  for (k = 0; k < 6; k++) {
    Y_tmp = k << 1;
    Y_tmp_0 = B[Y_tmp + r1];
    Y[Y_tmp + 1] = (B[Y_tmp + r2] - Y_tmp_0 * a21) / a22;
    Y[Y_tmp] = (Y_tmp_0 - Y[Y_tmp + 1] * a22_tmp) / A[r1];
  }
}

/* Function for MATLAB Function: '<S715>/MATLAB Function1' */
static real_T Gen2_ref_maximum_f5(const real_T x[7], struct Gen2* inst)
{
  real_T ex;
  int32_T idx;
  int32_T k;
  boolean_T exitg1;
  if (!rtIsNaN(x[0])) {
    idx = 1;
  } else {
    idx = 0;
    k = 2;
    exitg1 = false;
    while ((!exitg1) && (k < 8)) {
      if (!rtIsNaN(x[k - 1])) {
        idx = k;
        exitg1 = true;
      } else {
        k++;
      }
    }
  }

  if (idx == 0) {
    ex = x[0];
  } else {
    ex = x[idx - 1];
    while (idx + 1 <= 7) {
      if (ex < x[idx]) {
        ex = x[idx];
      }

      idx++;
    }
  }

  return ex;
}

/* Model step function */
void Gen2_ref_step(RT_MODEL_Gen2_ref *const Gen2_ref_M, struct Gen2* inst)
{
  struct BlockIO_Gen2_ref *Gen2_ref_B = Gen2_ref_M->blockIO;
  struct D_Work_Gen2_ref *Gen2_ref_DWork = Gen2_ref_M->dwork;
  struct PrevZCSigStates_Gen2_ref *Gen2_ref_PrevZCSigState = Gen2_ref_M->prevZCSigState;
  ExternalOutputs_Gen2_ref *Gen2_ref_Y = (ExternalOutputs_Gen2_ref *)
    Gen2_ref_M->outputs;

  /* local block i/o variables */
  real_T rtb_LookupTableDynamic2;
  real_T rtb_gainschedulingKeng1;
  real_T rtb_kappa0;
  real_T rtb_LookupTableDynamic;
  real_T rtb_LookupTableDynamic1;
  real_T rtb_gainschedulingKeng1_f;
  real_T rtb_CDSet_50;
  real_T rtb_CDSet_100;
  real_T rtb_LookupTableDynamic3;
  real_T rtb_LookupTableDynamic_n;
  real_T rtb_LookupTableDynamic_m;
  real_T rtb_LookupTableDynamic1_b;
  real_T rtb_gainschedulingKspeed;
  real_T rtb_gainschedulingTlam;
  real_T rtb_LookupTableDynamic2_h;
  real_T rtb_LookupTableDynamic_l;
  real_T rtb_LookupTableDynamic1_g;
  real_T rtb_gainschedulingD;
  real_T rtb_gainschedulingx_dist1;
  real_T rtb_gainschedulingKengPOW;
  real_T rtb_gainschedulingKeng;
  real_T rtb_LookupTableDynamic2_f;
  real_T rtb_LookupTableDynamic1_h;
  real_T rtb_LookupTableDynamic_h;
  real_T rtb_LookupTableDynamic_nk;
  real_T rtb_LookupTableDynamic1_o;
  real_T rtb_LookupTableDynamic_i;
  real_T rtb_LookupTableDynamic1_e;
  real_T rtb_LCRScal_Lam_EOT1;
  real_T rtb_LCRScal_Lam_EOT1_i;
  real_T rtb_Surgeprotectiondependingont;
  real_T rtb_Surgeprotectiondependingonb;
  real_T rtb_Lookup7;
  real_T rtb_Lookup6;
  real_T rtb_Lookup5;
  real_T rtb_Lookup4;
  real_T rtb_Lookup3;
  real_T rtb_Lookup2;
  real_T rtb_Lookup1;
  real_T rtb_kp_m;
  real_T u_lambda_past[100];
  real_T P_[36];
  real_T P_2inp_aug_tmp[36];
  real_T Phi_aug[36];
  real_T Phi_aug_0[36];
  real_T Phi_aug_1[36];
  real_T Phi_aug_2[36];
  real_T rtb_TmpSignalConversionAtSFunct[22];
  real_T Phi_obs_tmp_0[18];
  real_T rtb_K_KF_out[18];
  real_T R[16];
  real_T R_0[16];
  real_T rtb_ResettableDelay_br[13];
  real_T rtb_Switch3_je[13];
  real_T rtb_y_map_new[13];
  real_T rtb_y_map_new_n[13];
  real_T H_aug[12];
  real_T K_2inp_aug[12];
  real_T rtb_H_OUT[12];
  real_T rtb_H_OUT_0[12];
  real_T rtb_K_LQR[12];
  real_T rtb_K_LQR_0[12];
  real_T tmp[12];
  real_T rtb_Switch6_n[10];
  real_T B_d[9];
  real_T Phi_obs[9];
  real_T Q[9];
  real_T R_KF[9];
  real_T rtb_Phi_OUT[9];
  real_T rtb_Phi_OUT_0[9];
  real_T rtb_Phi_OUT_1[9];
  real_T rtb_Sum_og[8];
  real_T rtb_Switch_g[8];
  real_T rtb_Switch_dau[7];
  real_T rtb_y_map_new_a[7];
  real_T Hd_obs_0[6];
  real_T rtb_Switch_i5[6];
  real_T rtb_TmpSignalConversionAtDelayI[6];
  real_T rtb_TmpSignalConversionAtSFun_0[6];
  real_T rtb_TmpSignalConversionAtSFun_1[6];
  real_T x_[6];
  real_T rtb_Gain1_eu[5];
  real_T rtb_Gain2_k[5];
  real_T R_2inp[4];
  real_T rtb_Divide3_e[4];
  real_T rtb_Divide3_i0[4];
  real_T rtb_Divide_ab[4];
  real_T rtb_Product_m[4];
  real_T Hd_obs[3];
  real_T Phi_obs_tmp_1[3];
  real_T rtb_Switch1_cl[3];
  real_T rtb_TmpSignalConversionAtSFun_g[3];
  real_T rtb_TmpSignalConversionAtSFun_p[3];
  real_T rtb_err_KF[3];
  real_T rtb_err_cont[3];
  real_T rtb_TmpSignalConversionAtLoo_ht[2];
  real_T rtb_TmpSignalConversionAtLook_d[2];
  real_T rtb_u_sp_KF[2];
  real_T FILT_IN;
  real_T Ts_tmp;
  real_T delta_y;
  real_T delta_y_tmp_tmp;
  real_T err;
  real_T r;
  real_T rtb_Abs;
  real_T rtb_Abs_n;
  real_T rtb_Add2;
  real_T rtb_Add2_h;
  real_T rtb_BusCreator1_ref_P2_FB_CBV;
  real_T rtb_BusCreator1_ref_P2_FF;
  real_T rtb_BusCreator1_ref_P2s_FB_TV;
  real_T rtb_DataTypeConversion15;
  real_T rtb_DiscreteTimeIntegrator_g3;
  real_T rtb_Divide1_f1_tmp;
  real_T rtb_Divide1_fn;
  real_T rtb_Divide1_h4;
  real_T rtb_Divide1_k;
  real_T rtb_Divide2;
  real_T rtb_Divide2_a;
  real_T rtb_Divide2_f;
  real_T rtb_Divide3_a0;
  real_T rtb_Divide3_d;
  real_T rtb_Divide3_ep;
  real_T rtb_Divide3_g;
  real_T rtb_Divide3_k;
  real_T rtb_Divide3_n_tmp;
  real_T rtb_Divide3_p;
  real_T rtb_Divide4_d;
  real_T rtb_Divide4_ia;
  real_T rtb_Divide5_h;
  real_T rtb_Divide6_n;
  real_T rtb_Divide_br;
  real_T rtb_Divide_i1;
  real_T rtb_Divide_kp;
  real_T rtb_Divide_kt;
  real_T rtb_Divide_mr_tmp;
  real_T rtb_Divide_n0;
  real_T rtb_Gain;
  real_T rtb_Gain1_f_tmp;
  real_T rtb_Gain1_fr;
  real_T rtb_Gain1_o;
  real_T rtb_Gain2_ao;
  real_T rtb_Gain2_cm;
  real_T rtb_Gain3;
  real_T rtb_Gain6_b;
  real_T rtb_Gain6_jx;
  real_T rtb_Gain7;
  real_T rtb_Gain_i;
  real_T rtb_Gain_kl;
  real_T rtb_Gain_kp;
  real_T rtb_LogicalOperator1_js_tmp;
  real_T rtb_MassFlowCalc;
  real_T rtb_MinMax1_g;
  real_T rtb_MinMax1_h;
  real_T rtb_MinMax3;
  real_T rtb_MinMax_a;
  real_T rtb_MinMax_mf;
  real_T rtb_MinMax_n;
  real_T rtb_MultiportSwitch;
  real_T rtb_Pa2bar;
  real_T rtb_Pa2bar_k;
  real_T rtb_Pa2bar_o;
  real_T rtb_PactOut;
  real_T rtb_PactOut_o;
  real_T rtb_PactOut_tmp;
  real_T rtb_PrefOut;
  real_T rtb_Product1;
  real_T rtb_Product1_aq;
  real_T rtb_Product1_b;
  real_T rtb_Product1_b4;
  real_T rtb_Product1_bc;
  real_T rtb_Product1_c1_tmp;
  real_T rtb_Product1_e_tmp;
  real_T rtb_Product1_fu;
  real_T rtb_Product1_mqz;
  real_T rtb_Product2;
  real_T rtb_Product3_g;
  real_T rtb_Product4;
  real_T rtb_Product4_d;
  real_T rtb_Product_gj;
  real_T rtb_Product_l0;
  real_T rtb_Product_o;
  real_T rtb_RoundingFunction;
  real_T rtb_Saturation;
  real_T rtb_Saturation1_i;
  real_T rtb_Saturation6;
  real_T rtb_Saturation6_tmp;
  real_T rtb_Saturation_cx;
  real_T rtb_Saturation_e;
  real_T rtb_Saturation_gh;
  real_T rtb_Saturation_o;
  real_T rtb_Sum10;
  real_T rtb_Sum11;
  real_T rtb_Sum1_dh;
  real_T rtb_Sum1_idx_2;
  real_T rtb_Sum1_idx_3;
  real_T rtb_Sum1_jz;
  real_T rtb_Sum1_l;
  real_T rtb_Sum1_lo;
  real_T rtb_Sum2_a1;
  real_T rtb_Sum2_a_tmp;
  real_T rtb_Sum2_kg;
  real_T rtb_Sum3_hx;
  real_T rtb_Sum3_o;
  real_T rtb_Sum4_g;
  real_T rtb_Sum4_ny;
  real_T rtb_Sum5_iu;
  real_T rtb_Sum5_j;
  real_T rtb_Sum6_o_tmp;
  real_T rtb_Sum7_l5;
  real_T rtb_Sum8_m;
  real_T rtb_Sum_c;
  real_T rtb_Sum_e;
  real_T rtb_Sum_gb;
  real_T rtb_Sum_ig;
  real_T rtb_Sum_mf;
  real_T rtb_SumofElements;
  real_T rtb_SumofElements_l;
  real_T rtb_Switch13;
  real_T rtb_Switch1_d2;
  real_T rtb_Switch1_ep;
  real_T rtb_Switch1_k;
  real_T rtb_Switch1_kk;
  real_T rtb_Switch1_lk;
  real_T rtb_Switch1_mm;
  real_T rtb_Switch2_a;
  real_T rtb_Switch2_ba;
  real_T rtb_Switch2_by;
  real_T rtb_Switch2_c4;
  real_T rtb_Switch2_d1;
  real_T rtb_Switch2_ejy_tmp;
  real_T rtb_Switch2_ejy_tmp_0;
  real_T rtb_Switch2_g3;
  real_T rtb_Switch2_gd_idx_0;
  real_T rtb_Switch2_gd_idx_1;
  real_T rtb_Switch2_gd_idx_2;
  real_T rtb_Switch2_gd_idx_3;
  real_T rtb_Switch2_gs;
  real_T rtb_Switch2_h1;
  real_T rtb_Switch2_j0;
  real_T rtb_Switch2_jf;
  real_T rtb_Switch2_jq;
  real_T rtb_Switch2_jw;
  real_T rtb_Switch2_l;
  real_T rtb_Switch2_lu;
  real_T rtb_Switch2_n5;
  real_T rtb_Switch2_oou;
  real_T rtb_Switch4_p;
  real_T rtb_Switch5_iq;
  real_T rtb_Switch5_nn;
  real_T rtb_Switch8;
  real_T rtb_Switch9_k;
  real_T rtb_Switch_bs;
  real_T rtb_Switch_ct_tmp;
  real_T rtb_Switch_czo;
  real_T rtb_Switch_dhr;
  real_T rtb_Switch_dz_tmp;
  real_T rtb_Switch_e;
  real_T rtb_Switch_e3;
  real_T rtb_Switch_ed;
  real_T rtb_Switch_eu;
  real_T rtb_Switch_fi;
  real_T rtb_Switch_iy;
  real_T rtb_Switch_jv;
  real_T rtb_Switch_jz;
  real_T rtb_Switch_kr;
  real_T rtb_Switch_ks;
  real_T rtb_Switch_n;
  real_T rtb_Switch_nb;
  real_T rtb_Switch_on;
  real_T rtb_UkYk1_a4;
  real_T rtb_VariableIntegerDelay;
  real_T rtb_VariableIntegerDelay_b;
  real_T rtb_W2kW_o;
  real_T rtb_bResetHlci_0;
  real_T rtb_bar2Pa6;
  real_T rtb_deltafalllimit_ca;
  real_T rtb_deltafalllimit_h0;
  real_T rtb_dm_e;
  real_T rtb_dm_e_tmp;
  real_T rtb_etaBreakConst;
  real_T rtb_etaVolConst_lt;
  real_T rtb_kW2W;
  real_T rtb_kW2W1_h;
  real_T rtb_mbar2pa_g;
  real_T rtb_mbar2pa_i;
  real_T rtb_p1HP;
  real_T rtb_p1LP;
  real_T rtb_p2HP;
  real_T rtb_p2s;
  real_T rtb_rKK2_k;
  real_T rtb_rSkip_level;
  real_T rtb_up;
  real_T rtb_x_KF_out_idx_0;
  real_T rtb_x_KF_out_idx_1;
  real_T rtb_x_KF_out_idx_2;
  real_T rtb_x_sp_KF_idx_0;
  real_T rtb_x_sp_KF_idx_1;
  real_T rtb_x_sp_KF_idx_2;
  real_T u0;
  real_T u1;
  real_T x;
  real_T y_map_tmp;
  real_T y_map_tmp_0;
  int32_T Phi_aug_tmp;
  int32_T Phi_aug_tmp_0;
  int32_T i;
  int32_T k;
  int32_T rtb_H_OUT_tmp;
  int32_T rtb_K_LQR_tmp;
  real32_T rtb_BusCreator1_h_ui;
  real32_T rtb_TOF2_PT;
  real32_T rtb_rPos_CBV3;
  int16_T Npred;
  int16_T tmp_0;
  uint16_T rtb_DataTypeConversion_l;
  int8_T Phi_obs_tmp[18];
  uint8_T u0_0;
  boolean_T rtb_Act;
  boolean_T rtb_LogicalOperator;
  boolean_T rtb_LogicalOperator12_a;
  boolean_T rtb_LogicalOperator1_a0;
  boolean_T rtb_LogicalOperator1_e;
  boolean_T rtb_LogicalOperator1_i2;
  boolean_T rtb_LogicalOperator1_ix;
  boolean_T rtb_LogicalOperator1_j;
  boolean_T rtb_LogicalOperator1_ja;
  boolean_T rtb_LogicalOperator1_pa;
  boolean_T rtb_LogicalOperator2_dc;
  boolean_T rtb_LogicalOperator2_e;
  boolean_T rtb_LogicalOperator2_fy;
  boolean_T rtb_LogicalOperator2_k_tmp;
  boolean_T rtb_LogicalOperator2_l;
  boolean_T rtb_LogicalOperator2_ov;
  boolean_T rtb_LogicalOperator2_p1;
  boolean_T rtb_LogicalOperator3_aa;
  boolean_T rtb_LogicalOperator3_b;
  boolean_T rtb_LogicalOperator3_fj;
  boolean_T rtb_LogicalOperator3_gq;
  boolean_T rtb_LogicalOperator3_ja;
  boolean_T rtb_LogicalOperator3_k;
  boolean_T rtb_LogicalOperator4_go;
  boolean_T rtb_LogicalOperator4_m5;
  boolean_T rtb_LogicalOperator5;
  boolean_T rtb_LogicalOperator5_g_tmp;
  boolean_T rtb_LogicalOperator5_mv;
  boolean_T rtb_LogicalOperator5_p;
  boolean_T rtb_LogicalOperator_aw;
  boolean_T rtb_LogicalOperator_b;
  boolean_T rtb_LogicalOperator_cn;
  boolean_T rtb_LogicalOperator_f;
  boolean_T rtb_LogicalOperator_hi;
  boolean_T rtb_LogicalOperator_i;
  boolean_T rtb_LogicalOperator_in;
  boolean_T rtb_RelationalOperator1_j;
  boolean_T rtb_RelationalOperator2_j;
  boolean_T rtb_RelationalOperator_a;
  boolean_T rtb_RelationalOperator_l5;
  boolean_T rtb_RelationalOperator_ok;
  boolean_T rtb_Switch2_au;
  boolean_T rtb_Switch2_ij;
  boolean_T rtb_Switch2_jv;
  boolean_T rtb_Switch3_le;
  boolean_T rtb_Switch3_of;
  boolean_T rtb_Switch4_j;
  boolean_T rtb_Switch4_mu;
  boolean_T rtb_TOF_IN;
  boolean_T rtb_bActGasQualImprov;
  boolean_T rtb_bCBV_min;
  boolean_T rtb_bResetBdc;
  boolean_T rtb_bResetHlci;
  boolean_T rtb_bTV_sat;
  boolean_T rtb_bTriger_IT_LJ;
  boolean_T rtb_dbg_HLCi;
  boolean_T rtb_i_reset;
  static const int8_T b[18] = { 0, 0, 0, 0, 0, 0, 0, 0, 0, 1, 0, 0, 0, 1, 0, 0,
    0, 1 };

  static const real_T c[36] = { 0.0001, 0.0, 0.0, 0.0, 0.0, 0.0, 0.0, 0.0001,
    0.0, 0.0, 0.0, 0.0, 0.0, 0.0, 0.0001, 0.0, 0.0, 0.0, 0.0, 0.0, 0.0, 0.0001,
    0.0, 0.0, 0.0, 0.0, 0.0, 0.0, 0.0001, 0.0, 0.0, 0.0, 0.0, 0.0, 0.0, 0.0001 };

  static const int8_T C_aug[18] = { 1, 0, 0, 0, 1, 0, 0, 0, 1, 0, 0, 0, 0, 0, 0,
    0, 0, 0 };

  static const int8_T d[18] = { 1, 0, 0, 0, 0, 0, 0, 1, 0, 0, 0, 0, 0, 0, 1, 0,
    0, 0 };

  static const int8_T b_a[9] = { 1, 0, 0, 0, 1, 0, 0, 0, 1 };

  real_T rtb_Divide_mr_tmp_0;
  real_T rtb_Switch_fy_tmp_tmp;
  boolean_T exitg1;

  /* S-Function (bur_bus_in): '<Root>/Bus Input' */
  Gen2_ref_B->BusInput = inst->IN;

  /* Logic: '<S4>/Logical Operator' incorporates:
   *  Constant: '<S188>/Constant'
   *  RelationalOperator: '<S188>/Compare'
   */
  rtb_LogicalOperator = ((Gen2_ref_B->BusInput.iOpMode == 50) &&
    Gen2_ref_B->BusInput.bGen2_NetP_ena);

  /* S-Function (bur_bus_in): '<Root>/Bus Input3' */
  Gen2_ref_B->BusInput3 = inst->Para;

  /* Switch: '<S427>/Switch5' incorporates:
   *  Delay: '<S427>/Delay'
   *  RelationalOperator: '<S427>/Relational Operator11'
   */
  if (Gen2_ref_DWork->Delay_DSTATE[0] >=
      Gen2_ref_B->BusInput3.LR.rP_LR_Trig_GasStop_HL) {
    rtb_Divide4_d = Gen2_ref_B->BusInput3.LR.rP_LR_Trig_GasStop_HL;
  } else {
    rtb_Divide4_d = Gen2_ref_B->BusInput3.LR.rP_LR_Trig_GasStop;
  }

  /* End of Switch: '<S427>/Switch5' */

  /* RelationalOperator: '<S427>/Relational Operator13' incorporates:
   *  Delay: '<S427>/Delay'
   */
  rtb_LogicalOperator5_mv = (Gen2_ref_DWork->Delay_DSTATE[0] >= rtb_Divide4_d);

  /* Gain: '<S418>/Gain' incorporates:
   *  DataTypeConversion: '<S4>/Data Type Conversion34'
   */
  rtb_Gain = 0.10471975511965977 * Gen2_ref_B->BusInput.rN_Eng_LRskipF;

  /* Logic: '<S4>/Logical Operator8' incorporates:
   *  Constant: '<S189>/Constant'
   *  RelationalOperator: '<S189>/Compare'
   */
  rtb_bResetBdc = ((Gen2_ref_B->BusInput.iOpMode <= 10) ||
                   Gen2_ref_B->BusInput.bResetGlobal);

  /* Logic: '<S4>/Logical Operator5' incorporates:
   *  Constant: '<S187>/Constant'
   *  Logic: '<S4>/Logical Operator1'
   *  Logic: '<S4>/Logical Operator4'
   *  RelationalOperator: '<S187>/Compare'
   */
  rtb_bResetHlci = (rtb_bResetBdc || ((Gen2_ref_B->BusInput.iOpMode != 60) ||
    (!Gen2_ref_B->BusInput.bGen2_island_ena)));

  /* Outputs for Atomic SubSystem: '<S418>/2nd Order Filter' */
  Gen2_ref_undOrderFilter3(rtb_Gain,
    Gen2_ref_B->BusInput3.SpeedCtrl.r2ndOrdFiltOmega_N_Prot,
    Gen2_ref_B->BusInput3.SpeedCtrl.r2ndOrdFiltD_N_Prot, rtb_bResetHlci,
    &Gen2_ref_B->undOrderFilter_j, &Gen2_ref_DWork->undOrderFilter_j, inst);

  /* End of Outputs for SubSystem: '<S418>/2nd Order Filter' */

  /* Outputs for Atomic SubSystem: '<S418>/Filter' */
  /* RelationalOperator: '<S439>/Relational Operator' incorporates:
   *  Constant: '<S439>/Constant'
   */
  rtb_bCBV_min = (Gen2_ref_B->BusInput3.SpeedCtrl.rTi_Prot > 0.0);

  /* Logic: '<S439>/Logical Operator' incorporates:
   *  Logic: '<S439>/Logical Operator1'
   */
  rtb_LogicalOperator_in = (rtb_bResetHlci || (!rtb_bCBV_min));

  /* DiscreteIntegrator: '<S439>/Discrete-Time Integrator' */
  if (Gen2_ref_DWork->DiscreteTimeIntegrator_IC_LOA_f != 0) {
    Gen2_ref_DWork->DiscreteTimeIntegrator_DSTAT_eh = rtb_Gain;
  }

  if (rtb_LogicalOperator_in || (Gen2_ref_DWork->DiscreteTimeIntegrator_PrevRe_g
       != 0)) {
    Gen2_ref_DWork->DiscreteTimeIntegrator_DSTAT_eh = rtb_Gain;
  }

  /* Abs: '<S442>/Abs' */
  FILT_IN = fabs(Gen2_ref_B->BusInput3.SpeedCtrl.rTi_Prot);

  /* Switch: '<S442>/Switch' incorporates:
   *  Constant: '<S442>/Constant2'
   *  RelationalOperator: '<S442>/Relational Operator'
   */
  if (2.2204460492503131E-16 >= FILT_IN) {
    rtb_bResetHlci_0 = 2.2204460492503131E-16;
  } else {
    rtb_bResetHlci_0 = Gen2_ref_B->BusInput3.SpeedCtrl.rTi_Prot;
  }

  /* End of Switch: '<S442>/Switch' */

  /* Product: '<S439>/Divide4' incorporates:
   *  DiscreteIntegrator: '<S439>/Discrete-Time Integrator'
   *  Sum: '<S439>/Sum4'
   */
  rtb_Divide4_ia = (rtb_Gain - Gen2_ref_DWork->DiscreteTimeIntegrator_DSTAT_eh) /
    rtb_bResetHlci_0;

  /* Switch: '<S439>/Switch' incorporates:
   *  DiscreteIntegrator: '<S439>/Discrete-Time Integrator'
   */
  if (rtb_bCBV_min) {
    rtb_Switch_ed = Gen2_ref_DWork->DiscreteTimeIntegrator_DSTAT_eh;
  } else {
    rtb_Switch_ed = rtb_Gain;
  }

  /* End of Switch: '<S439>/Switch' */

  /* Update for DiscreteIntegrator: '<S439>/Discrete-Time Integrator' */
  Gen2_ref_DWork->DiscreteTimeIntegrator_IC_LOA_f = 0U;
  Gen2_ref_DWork->DiscreteTimeIntegrator_DSTAT_eh += 0.01 * rtb_Divide4_ia;
  Gen2_ref_DWork->DiscreteTimeIntegrator_PrevRe_g = (int8_T)
    rtb_LogicalOperator_in;

  /* End of Outputs for SubSystem: '<S418>/Filter' */

  /* Switch: '<S418>/Switch' incorporates:
   *  Switch: '<S418>/Switch1'
   */
  if (Gen2_ref_B->BusInput3.SpeedCtrl.b2ndOrdFilt_N_Prot) {
    rtb_Switch_eu = Gen2_ref_B->undOrderFilter_j.Switch;
    rtb_Switch1_mm = Gen2_ref_B->undOrderFilter_j.Switch1;
  } else {
    rtb_Switch_eu = rtb_Switch_ed;

    /* Outputs for Atomic SubSystem: '<S418>/Filter' */
    /* Switch: '<S439>/Switch1' incorporates:
     *  Constant: '<S439>/Constant'
     */
    if (rtb_LogicalOperator_in) {
      rtb_Switch1_mm = 0.0;
    } else {
      rtb_Switch1_mm = rtb_Divide4_ia;
    }

    /* End of Switch: '<S439>/Switch1' */
    /* End of Outputs for SubSystem: '<S418>/Filter' */
  }

  /* End of Switch: '<S418>/Switch' */

  /* Gain: '<S418>/Gain1' incorporates:
   *  Product: '<S418>/Divide'
   */
  rtb_Gain1_fr = -(rtb_Switch_eu * rtb_Switch1_mm *
                   Gen2_ref_B->BusInput3.eng.rJ_Eng);

  /* Abs: '<S508>/Abs' incorporates:
   *  Abs: '<S605>/Abs'
   *  Abs: '<S858>/Abs'
   */
  rtb_Product1_e_tmp = fabs(Gen2_ref_B->BusInput3.eng.rP_Nom);

  /* Switch: '<S508>/Switch' incorporates:
   *  Abs: '<S508>/Abs'
   *  Constant: '<S508>/Constant2'
   *  RelationalOperator: '<S508>/Relational Operator'
   */
  if (2.2204460492503131E-16 >= rtb_Product1_e_tmp) {
    rtb_bResetHlci_0 = 2.2204460492503131E-16;
  } else {
    rtb_bResetHlci_0 = Gen2_ref_B->BusInput3.eng.rP_Nom;
  }

  /* End of Switch: '<S508>/Switch' */

  /* Gain: '<S427>/Gain6' incorporates:
   *  Gain: '<S427>/Gain2'
   *  Product: '<S427>/Divide3'
   */
  rtb_Saturation = -(0.001 * rtb_Gain1_fr / rtb_bResetHlci_0);

  /* Saturate: '<S427>/Saturation' */
  if (rtb_Saturation > 1000.0) {
    rtb_Saturation = 1000.0;
  } else if (rtb_Saturation < 0.0) {
    rtb_Saturation = 0.0;
  }

  /* End of Saturate: '<S427>/Saturation' */

  /* RelationalOperator: '<S427>/Relational Operator8' */
  rtb_dbg_HLCi = (rtb_Saturation > rtb_Divide4_d);

  /* DataTypeConversion: '<S4>/Data Type Conversion15' */
  rtb_DataTypeConversion15 = Gen2_ref_B->BusInput.rN_Eng;

  /* Outputs for Atomic SubSystem: '<S201>/Volt_filt' */
  /* DataTypeConversion: '<S4>/Data Type Conversion17' */
  Gen2_ref_N_TC_HP_filt((real_T)Gen2_ref_B->BusInput.rU_Gen_Norm,
                        Gen2_ref_B->BusInput3.inFilt.rTiF_V, rtb_bResetBdc,
                        &Gen2_ref_B->Volt_filt, &Gen2_ref_DWork->Volt_filt, inst);

  /* End of Outputs for SubSystem: '<S201>/Volt_filt' */

  /* Gain: '<S4>/Gain2' incorporates:
   *  DataTypeConversion: '<S4>/Data Type Conversion13'
   */
  rtb_Gain2_ao = 1000.0 * Gen2_ref_B->BusInput.rP_Act;

  /* Gain: '<S4>/kW2W' incorporates:
   *  DataTypeConversion: '<S4>/Data Type Conversion19'
   */
  rtb_kW2W = 1000.0 * Gen2_ref_B->BusInput.rP_Set;

  /* Gain: '<S4>/bar2Pa3' incorporates:
   *  DataTypeConversion: '<S4>/Data Type Conversion5'
   */
  rtb_p2s = 100000.0 * Gen2_ref_B->BusInput.tPr.rp2s;

  /* Outputs for Atomic SubSystem: '<S205>/p2s_filt' */
  Gen2_ref_N_TC_HP_filt(rtb_p2s, Gen2_ref_B->BusInput3.inFilt.rTiF_Pr,
                        rtb_bResetBdc, &Gen2_ref_B->p2s_filt,
                        &Gen2_ref_DWork->p2s_filt, inst);

  /* End of Outputs for SubSystem: '<S205>/p2s_filt' */

  /* SignalConversion generated from: '<S425>/Delay' incorporates:
   *  DataTypeConversion: '<S4>/Data Type Conversion16'
   */
  rtb_TmpSignalConversionAtDelayI[0] = rtb_DataTypeConversion15;
  rtb_TmpSignalConversionAtDelayI[1] = Gen2_ref_B->BusInput.rN_Set;
  rtb_TmpSignalConversionAtDelayI[2] = Gen2_ref_B->Volt_filt.Switch;
  rtb_TmpSignalConversionAtDelayI[3] = rtb_Gain2_ao;
  rtb_TmpSignalConversionAtDelayI[4] = rtb_kW2W;

  /* Switch: '<S8>/Switch7' */
  if (Gen2_ref_B->BusInput3.SpeedCtrl.bUseFilteredFeedback) {
    /* SignalConversion generated from: '<S425>/Delay' */
    rtb_TmpSignalConversionAtDelayI[5] = Gen2_ref_B->p2s_filt.Switch;
  } else {
    /* SignalConversion generated from: '<S425>/Delay' */
    rtb_TmpSignalConversionAtDelayI[5] = rtb_p2s;
  }

  /* End of Switch: '<S8>/Switch7' */

  /* Delay: '<S425>/Delay' incorporates:
   *  Switch: '<S425>/Switch'
   */
  Gen2_ref_DWork->icLoad = ((((Gen2_ref_PrevZCSigState->Delay_Reset_ZCE == 1) !=
    (int32_T)rtb_bResetHlci) && (Gen2_ref_PrevZCSigState->Delay_Reset_ZCE != 3))
    || rtb_bResetHlci || Gen2_ref_DWork->icLoad);
  Gen2_ref_PrevZCSigState->Delay_Reset_ZCE = rtb_bResetHlci;
  for (i = 0; i < 6; i++) {
    rtb_Divide4_d = rtb_TmpSignalConversionAtDelayI[i];
    if (Gen2_ref_DWork->icLoad) {
      Gen2_ref_DWork->Delay_DSTATE_o[i] = rtb_Divide4_d;
    }

    /* Switch: '<S425>/Switch' */
    if (Gen2_ref_B->BusInput.tLvrt.bLvrtFlg) {
      rtb_Divide4_d = Gen2_ref_DWork->Delay_DSTATE_o[i];
    }

    rtb_TmpSignalConversionAtDelayI[i] = rtb_Divide4_d;
  }

  /* Outputs for Atomic SubSystem: '<S425>/TOF' */
  /* Constant: '<S425>/Constant3' */
  Gen2_ref_TOF(Gen2_ref_B->BusInput.tLvrt.bLvrtFlg, 1.0, &Gen2_ref_B->TOF_h,
               &Gen2_ref_DWork->TOF_h, inst);

  /* End of Outputs for SubSystem: '<S425>/TOF' */

  /* Logic: '<S425>/Logical Operator2' incorporates:
   *  Logic: '<S26>/Logical Operator2'
   *  Logic: '<S45>/Logical Operator2'
   */
  rtb_LogicalOperator_b = !Gen2_ref_B->BusInput.tLvrt.bLvrtFlg;

  /* Outputs for Atomic SubSystem: '<S425>/Filter' */
  /* Logic: '<S485>/Logical Operator' incorporates:
   *  Logic: '<S425>/Logical Operator1'
   *  Logic: '<S425>/Logical Operator2'
   *  Logic: '<S425>/Logical Operator3'
   */
  rtb_LogicalOperator_in = (((!Gen2_ref_B->TOF_h.LogicalOperator1) &&
    rtb_LogicalOperator_b) || rtb_bResetHlci ||
    Gen2_ref_B->BusInput3.SpeedCtrl.bReset_LVRT_inputFilter);

  /* DiscreteIntegrator: '<S485>/Discrete-Time Integrator' */
  if (Gen2_ref_DWork->DiscreteTimeIntegrator_IC_LOA_p != 0) {
    for (i = 0; i < 6; i++) {
      Gen2_ref_DWork->DiscreteTimeIntegrator_DSTAT_gl[i] =
        rtb_TmpSignalConversionAtDelayI[i];
    }
  }

  /* Update for DiscreteIntegrator: '<S485>/Discrete-Time Integrator' */
  Gen2_ref_DWork->DiscreteTimeIntegrator_IC_LOA_p = 0U;
  for (i = 0; i < 6; i++) {
    /* Switch: '<S485>/Switch' */
    rtb_Divide4_d = rtb_TmpSignalConversionAtDelayI[i];

    /* DiscreteIntegrator: '<S485>/Discrete-Time Integrator' */
    if (rtb_LogicalOperator_in ||
        (Gen2_ref_DWork->DiscreteTimeIntegrator_PrevR_cs != 0)) {
      Gen2_ref_DWork->DiscreteTimeIntegrator_DSTAT_gl[i] = rtb_Divide4_d;
    }

    /* Switch: '<S485>/Switch' incorporates:
     *  DiscreteIntegrator: '<S485>/Discrete-Time Integrator'
     */
    rtb_Switch_i5[i] = Gen2_ref_DWork->DiscreteTimeIntegrator_DSTAT_gl[i];

    /* Update for DiscreteIntegrator: '<S485>/Discrete-Time Integrator' incorporates:
     *  Product: '<S485>/Divide4'
     *  Sum: '<S485>/Sum4'
     */
    Gen2_ref_DWork->DiscreteTimeIntegrator_DSTAT_gl[i] += (rtb_Divide4_d -
      Gen2_ref_DWork->DiscreteTimeIntegrator_DSTAT_gl[i]) / 0.1 * 0.01;
  }

  /* Update for DiscreteIntegrator: '<S485>/Discrete-Time Integrator' */
  Gen2_ref_DWork->DiscreteTimeIntegrator_PrevR_cs = (int8_T)
    rtb_LogicalOperator_in;

  /* End of Outputs for SubSystem: '<S425>/Filter' */

  /* Switch: '<S424>/Switch' */
  if (Gen2_ref_B->BusInput3.SpeedCtrl.bLSLdeactNref) {
    rtb_Switch_ks = Gen2_ref_B->BusInput3.eng.rN_Nom;
  } else {
    rtb_Switch_ks = rtb_Switch_i5[1];
  }

  /* End of Switch: '<S424>/Switch' */

  /* Switch: '<S509>/Switch' incorporates:
   *  Abs: '<S509>/Abs'
   *  Constant: '<S509>/Constant2'
   *  RelationalOperator: '<S509>/Relational Operator'
   */
  if (2.2204460492503131E-16 >= fabs(rtb_Switch_ks)) {
    rtb_bResetHlci_0 = 2.2204460492503131E-16;
  } else {
    rtb_bResetHlci_0 = rtb_Switch_ks;
  }

  /* End of Switch: '<S509>/Switch' */

  /* Product: '<S427>/Divide4' incorporates:
   *  DataTypeConversion: '<S4>/Data Type Conversion34'
   */
  rtb_Divide4_d = Gen2_ref_B->BusInput.rN_Eng_LRskipF / rtb_bResetHlci_0;

  /* RelationalOperator: '<S427>/Relational Operator3' */
  rtb_RelationalOperator2_j = (rtb_Divide4_d >
    Gen2_ref_B->BusInput3.LR.rN_LR_Trig_GasStop);
```
